(* IEC 61131-3 sources: inproshop/Team-Test5_exported/2.Main, 7 files *)

(* ---- Main.ST ---- *)
(* ==== Generated by PlcOpcUaHmi at 2026-04-27 16:09:01  source=DB80_IO ==== *)
VAR_GLOBAL
	IX8000_0	AT	%IX8000.0:BOOL;
	IX8000_1	AT	%IX8000.1:BOOL;
	IX8000_2	AT	%IX8000.2:BOOL;
	IX8000_3	AT	%IX8000.3:BOOL;
	IX8000_4	AT	%IX8000.4:BOOL;
	IX8000_5	AT	%IX8000.5:BOOL;
	IX8000_6	AT	%IX8000.6:BOOL;
	IX8000_7	AT	%IX8000.7:BOOL;
	IX8001_0_OP08启动按钮HMI1	AT	%IX8001.0:BOOL;
	IX8001_1_OP08停止按钮HMI	AT	%IX8001.1:BOOL;
	IX8001_2_OP08复位按钮HMI	AT	%IX8001.2:BOOL;
	IX8001_3_OP08手自动旋钮HMI	AT	%IX8001.3:BOOL;
	IX8001_4_OP08急停按钮HMI	AT	%IX8001.4:BOOL;
	IX8001_5_OP08启动按钮左	AT	%IX8001.5:BOOL;
	IX8001_6_OP08停止按钮左	AT	%IX8001.6:BOOL;
	IX8001_7_OP08复位按钮左	AT	%IX8001.7:BOOL;
	IX8002_0_OP08手自动旋钮左	AT	%IX8002.0:BOOL;
	IX8002_1_OP08急停按钮左	AT	%IX8002.1:BOOL;
	IX8002_2_OP08启动按钮右	AT	%IX8002.2:BOOL;
	IX8002_3_OP08停止按钮右	AT	%IX8002.3:BOOL;
	IX8002_4_OP08复位按钮右	AT	%IX8002.4:BOOL;
	IX8002_5_OP08手自动旋钮右	AT	%IX8002.5:BOOL;
	IX8002_6_OP08急停按钮右	AT	%IX8002.6:BOOL;
	IX8002_7_OP08安全门1	AT	%IX8002.7:BOOL;
	IX8003_0_OP08安全门2	AT	%IX8003.0:BOOL;
	IX8003_1_OP08安全门3	AT	%IX8003.1:BOOL;
	IX8003_2_OP08安全门4	AT	%IX8003.2:BOOL;
	IX8003_3_OP08安全门5	AT	%IX8003.3:BOOL;
	IX8003_4_OP08安全门6	AT	%IX8003.4:BOOL;
	IX8003_5_OP08安全门7	AT	%IX8003.5:BOOL;
	IX8003_6_OP08安全门8	AT	%IX8003.6:BOOL;
	IX8003_7	AT	%IX8003.7:BOOL;
	IX8004_0	AT	%IX8004.0:BOOL;
	IX8004_1	AT	%IX8004.1:BOOL;
	IX8004_2	AT	%IX8004.2:BOOL;
	IX8004_3	AT	%IX8004.3:BOOL;
	IX8004_4	AT	%IX8004.4:BOOL;
	IX8004_5	AT	%IX8004.5:BOOL;
	IX8004_6	AT	%IX8004.6:BOOL;
	IX8004_7	AT	%IX8004.7:BOOL;
	IX8005_0	AT	%IX8005.0:BOOL;
	IX8005_1	AT	%IX8005.1:BOOL;
	IX8005_2	AT	%IX8005.2:BOOL;
	IX8005_3	AT	%IX8005.3:BOOL;
	IX8005_4	AT	%IX8005.4:BOOL;
	IX8005_5	AT	%IX8005.5:BOOL;
	IX8005_6	AT	%IX8005.6:BOOL;
	IX8005_7	AT	%IX8005.7:BOOL;
	IX8006_0	AT	%IX8006.0:BOOL;
	IX8006_1	AT	%IX8006.1:BOOL;
	IX8006_2	AT	%IX8006.2:BOOL;
	IX8006_3	AT	%IX8006.3:BOOL;
	IX8006_4	AT	%IX8006.4:BOOL;
	IX8006_5	AT	%IX8006.5:BOOL;
	IX8006_6	AT	%IX8006.6:BOOL;
	IX8006_7	AT	%IX8006.7:BOOL;
	IX8007_0	AT	%IX8007.0:BOOL;
	IX8007_1	AT	%IX8007.1:BOOL;
	IX8007_2	AT	%IX8007.2:BOOL;
	IX8007_3	AT	%IX8007.3:BOOL;
	IX8007_4	AT	%IX8007.4:BOOL;
	IX8007_5	AT	%IX8007.5:BOOL;
	IX8007_6	AT	%IX8007.6:BOOL;
	IX8007_7	AT	%IX8007.7:BOOL;
	IX8008_0	AT	%IX8008.0:BOOL;
	IX8008_1	AT	%IX8008.1:BOOL;
	IX8008_2	AT	%IX8008.2:BOOL;
	IX8008_3	AT	%IX8008.3:BOOL;
	IX8008_4	AT	%IX8008.4:BOOL;
	IX8008_5	AT	%IX8008.5:BOOL;
	IX8008_6	AT	%IX8008.6:BOOL;
	IX8008_7	AT	%IX8008.7:BOOL;
	IX8009_0	AT	%IX8009.0:BOOL;
	IX8009_1	AT	%IX8009.1:BOOL;
	IX8009_2	AT	%IX8009.2:BOOL;
	IX8009_3	AT	%IX8009.3:BOOL;
	IX8009_4	AT	%IX8009.4:BOOL;
	IX8009_5	AT	%IX8009.5:BOOL;
	IX8009_6	AT	%IX8009.6:BOOL;
	IX8009_7	AT	%IX8009.7:BOOL;
	IX8100_0_工位1_人工操作按钮	AT	%IX8100.0:BOOL;
	IX8100_1_工位1_物料到位感应Sensor1	AT	%IX8100.1:BOOL;
	IX8100_2_工位1_预留	AT	%IX8100.2:BOOL;
	IX8100_3_工位2_人工操作按钮	AT	%IX8100.3:BOOL;
	IX8100_4_工位2_物料到位感应Sensor2	AT	%IX8100.4:BOOL;
	IX8100_5_工位2_预留	AT	%IX8100.5:BOOL;
	IX8100_6_工位3_人工操作按钮	AT	%IX8100.6:BOOL;
	IX8100_7_工位3_物料到位感应Sensor3	AT	%IX8100.7:BOOL;
	IX8101_0_工位3_预留	AT	%IX8101.0:BOOL;
	IX8101_1_工位4_人工操作按钮	AT	%IX8101.1:BOOL;
	IX8101_2_工位4_物料到位感应Sensor4	AT	%IX8101.2:BOOL;
	IX8101_3_工位4_预留	AT	%IX8101.3:BOOL;
	IX8101_4_工位5_人工操作按钮	AT	%IX8101.4:BOOL;
	IX8101_5_工位5_物料到位感应Sensor5	AT	%IX8101.5:BOOL;
	IX8101_6_工位5_预留	AT	%IX8101.6:BOOL;
	IX8101_7_工位6_人工操作按钮	AT	%IX8101.7:BOOL;
	IX8102_0_工位6_物料到位感应Sensor6	AT	%IX8102.0:BOOL;
	IX8102_1_工位6_预留	AT	%IX8102.1:BOOL;
	IX8102_2_工位7_人工操作按钮	AT	%IX8102.2:BOOL;
	IX8102_3_工位7_物料到位感应Sensor7	AT	%IX8102.3:BOOL;
	IX8102_4_工位7_预留	AT	%IX8102.4:BOOL;
	IX8102_5_工位8_人工操作按钮	AT	%IX8102.5:BOOL;
	IX8102_6_工位8_物料到位感应Sensor8	AT	%IX8102.6:BOOL;
	IX8102_7_工位8_预留	AT	%IX8102.7:BOOL;
	IX8103_0_工位9_人工操作按钮	AT	%IX8103.0:BOOL;
	IX8103_1_工位9_物料到位感应Sensor9	AT	%IX8103.1:BOOL;
	IX8103_2_工位9_预留	AT	%IX8103.2:BOOL;
	IX8103_3_工位10_人工操作按钮	AT	%IX8103.3:BOOL;
	IX8103_4_工位10_物料到位感应Sensor10	AT	%IX8103.4:BOOL;
	IX8103_5_工位10_预留	AT	%IX8103.5:BOOL;
	IX8103_6	AT	%IX8103.6:BOOL;
	IX8103_7	AT	%IX8103.7:BOOL;
	IX8104_0_工位11_人工操作按钮	AT	%IX8104.0:BOOL;
	IX8104_1_工位11_物料到位感应Sensor11	AT	%IX8104.1:BOOL;
	IX8104_2_工位11_预留	AT	%IX8104.2:BOOL;
	IX8104_3_工位12_人工操作按钮	AT	%IX8104.3:BOOL;
	IX8104_4_工位12_物料到位感应Sensor12	AT	%IX8104.4:BOOL;
	IX8104_5_工位12_预留	AT	%IX8104.5:BOOL;
	IX8104_6_工位13_人工操作按钮	AT	%IX8104.6:BOOL;
	IX8104_7_工位13_物料到位感应Sensor13	AT	%IX8104.7:BOOL;
	IX8105_0_工位13_预留	AT	%IX8105.0:BOOL;
	IX8105_1_工位14_人工操作按钮	AT	%IX8105.1:BOOL;
	IX8105_2_工位14_物料到位感应Sensor14	AT	%IX8105.2:BOOL;
	IX8105_3_工位14_预留	AT	%IX8105.3:BOOL;
	IX8105_4_工位15_人工操作按钮	AT	%IX8105.4:BOOL;
	IX8105_5_工位15_物料到位感应Sensor15	AT	%IX8105.5:BOOL;
	IX8105_6_工位15_预留	AT	%IX8105.6:BOOL;
	IX8105_7_工位16_人工操作按钮	AT	%IX8105.7:BOOL;
	IX8106_0_工位16_物料到位感应Sensor16	AT	%IX8106.0:BOOL;
	IX8106_1_工位16_预留	AT	%IX8106.1:BOOL;
	IX8106_2_工位17_人工操作按钮	AT	%IX8106.2:BOOL;
	IX8106_3_工位17_物料到位感应Sensor17	AT	%IX8106.3:BOOL;
	IX8106_4_工位17_预留	AT	%IX8106.4:BOOL;
	IX8106_5_工位18_人工操作按钮	AT	%IX8106.5:BOOL;
	IX8106_6_工位18_物料到位感应Sensor18	AT	%IX8106.6:BOOL;
	IX8106_7_工位18_预留	AT	%IX8106.7:BOOL;
	IX8107_0_工位19_人工操作按钮	AT	%IX8107.0:BOOL;
	IX8107_1_工位19_物料到位感应Sensor19	AT	%IX8107.1:BOOL;
	IX8107_2_工位19_预留	AT	%IX8107.2:BOOL;
	IX8107_3_工位20_人工操作按钮	AT	%IX8107.3:BOOL;
	IX8107_4_工位20_物料到位感应Sensor20	AT	%IX8107.4:BOOL;
	IX8107_5_工位20_预留	AT	%IX8107.5:BOOL;
	IX8107_6	AT	%IX8107.6:BOOL;
	IX8107_7	AT	%IX8107.7:BOOL;
	IX8108_0_工位21_人工操作按钮	AT	%IX8108.0:BOOL;
	IX8108_1_工位21_物料到位感应Sensor21	AT	%IX8108.1:BOOL;
	IX8108_2_工位21_预留	AT	%IX8108.2:BOOL;
	IX8108_3_工位22_人工操作按钮	AT	%IX8108.3:BOOL;
	IX8108_4_工位22_物料到位感应Sensor22	AT	%IX8108.4:BOOL;
	IX8108_5_工位22_预留	AT	%IX8108.5:BOOL;
	IX8108_6_工位23_人工操作按钮	AT	%IX8108.6:BOOL;
	IX8108_7_工位23_物料到位感应Sensor23	AT	%IX8108.7:BOOL;
	IX8109_0_工位23_预留	AT	%IX8109.0:BOOL;
	IX8109_1_工位24_人工操作按钮	AT	%IX8109.1:BOOL;
	IX8109_2_工位24_物料到位感应Sensor24	AT	%IX8109.2:BOOL;
	IX8109_3_工位24_预留	AT	%IX8109.3:BOOL;
	IX8109_4_工位25_人工操作按钮	AT	%IX8109.4:BOOL;
	IX8109_5_工位25_物料到位感应Sensor25	AT	%IX8109.5:BOOL;
	IX8109_6_工位25_预留	AT	%IX8109.6:BOOL;
	IX8109_7_工位26_人工操作按钮	AT	%IX8109.7:BOOL;
	IX8110_0_工位26_物料到位感应Sensor26	AT	%IX8110.0:BOOL;
	IX8110_1_工位26_预留	AT	%IX8110.1:BOOL;
	IX8110_2_工位27_人工操作按钮	AT	%IX8110.2:BOOL;
	IX8110_3_工位27_物料到位感应Sensor27	AT	%IX8110.3:BOOL;
	IX8110_4_工位27_预留	AT	%IX8110.4:BOOL;
	IX8110_5_工位28_人工操作按钮	AT	%IX8110.5:BOOL;
	IX8110_6_工位28_物料到位感应Sensor28	AT	%IX8110.6:BOOL;
	IX8110_7_工位28_预留	AT	%IX8110.7:BOOL;
	IX8111_0_工位29_人工操作按钮	AT	%IX8111.0:BOOL;
	IX8111_1_工位29_物料到位感应Sensor29	AT	%IX8111.1:BOOL;
	IX8111_2_工位29_预留	AT	%IX8111.2:BOOL;
	IX8111_3_工位30_人工操作按钮	AT	%IX8111.3:BOOL;
	IX8111_4_工位30_物料到位感应Sensor30	AT	%IX8111.4:BOOL;
	IX8111_5_工位30_预留1	AT	%IX8111.5:BOOL;
	IX8111_6	AT	%IX8111.6:BOOL;
	IX8111_7	AT	%IX8111.7:BOOL;
	IX8112_0_工位31_人工操作按钮	AT	%IX8112.0:BOOL;
	IX8112_1_工位31_物料到位感应Sensor31	AT	%IX8112.1:BOOL;
	IX8112_2_工位31_预留	AT	%IX8112.2:BOOL;
	IX8112_3_工位32_人工操作按钮	AT	%IX8112.3:BOOL;
	IX8112_4_工位32_物料到位感应Sensor32	AT	%IX8112.4:BOOL;
	IX8112_5_工位32_预留	AT	%IX8112.5:BOOL;
	IX8112_6_工位33_人工操作按钮	AT	%IX8112.6:BOOL;
	IX8112_7_工位33_物料到位感应Sensor33	AT	%IX8112.7:BOOL;
	IX8113_0_工位33_预留	AT	%IX8113.0:BOOL;
	IX8113_1_工位34_人工操作按钮	AT	%IX8113.1:BOOL;
	IX8113_2_工位34_物料到位感应Sensor34	AT	%IX8113.2:BOOL;
	IX8113_3_工位34_预留	AT	%IX8113.3:BOOL;
	IX8113_4_工位35_人工操作按钮	AT	%IX8113.4:BOOL;
	IX8113_5_工位35_物料到位感应Sensor35	AT	%IX8113.5:BOOL;
	IX8113_6_工位35_预留	AT	%IX8113.6:BOOL;
	IX8113_7_工位36_人工操作按钮	AT	%IX8113.7:BOOL;
	IX8114_0_工位36_物料到位感应Sensor36	AT	%IX8114.0:BOOL;
	IX8114_1_工位36_预留	AT	%IX8114.1:BOOL;
	IX8114_2_工位37_人工操作按钮	AT	%IX8114.2:BOOL;
	IX8114_3_工位37_物料到位感应Sensor37	AT	%IX8114.3:BOOL;
	IX8114_4_工位37_预留	AT	%IX8114.4:BOOL;
	IX8114_5_工位38_人工操作按钮	AT	%IX8114.5:BOOL;
	IX8114_6_工位38_物料到位感应Sensor38	AT	%IX8114.6:BOOL;
	IX8114_7_工位38_预留	AT	%IX8114.7:BOOL;
	IX8115_0_工位39_人工操作按钮	AT	%IX8115.0:BOOL;
	IX8115_1_工位39_物料到位感应Sensor39	AT	%IX8115.1:BOOL;
	IX8115_2_工位39_预留	AT	%IX8115.2:BOOL;
	IX8115_3_工位40_人工操作按钮	AT	%IX8115.3:BOOL;
	IX8115_4_工位40_物料到位感应Sensor40	AT	%IX8115.4:BOOL;
	IX8115_5_工位40_预留	AT	%IX8115.5:BOOL;
	IX8115_6	AT	%IX8115.6:BOOL;
	IX8115_7	AT	%IX8115.7:BOOL;
	IX8200_0_工位41_人工操作按钮	AT	%IX8200.0:BOOL;
	IX8200_1_工位41_物料到位感应Sensor41	AT	%IX8200.1:BOOL;
	IX8200_2_工位41_预留	AT	%IX8200.2:BOOL;
	IX8200_3_工位42_人工操作按钮	AT	%IX8200.3:BOOL;
	IX8200_4_工位42_物料到位感应Sensor42	AT	%IX8200.4:BOOL;
	IX8200_5_工位42_预留	AT	%IX8200.5:BOOL;
	IX8200_6_工位43_人工操作按钮	AT	%IX8200.6:BOOL;
	IX8200_7_工位43_物料到位感应Sensor43	AT	%IX8200.7:BOOL;
	IX8201_0_工位43_预留	AT	%IX8201.0:BOOL;
	IX8201_1_工位44_人工操作按钮	AT	%IX8201.1:BOOL;
	IX8201_2_工位44_物料到位感应Sensor44	AT	%IX8201.2:BOOL;
	IX8201_3_工位44_预留	AT	%IX8201.3:BOOL;
	IX8201_4_工位45_人工操作按钮	AT	%IX8201.4:BOOL;
	IX8201_5_工位45_物料到位感应Sensor45	AT	%IX8201.5:BOOL;
	IX8201_6_工位45_预留	AT	%IX8201.6:BOOL;
	IX8201_7_工位46_人工操作按钮	AT	%IX8201.7:BOOL;
	IX8202_0_工位46_物料到位感应Sensor46	AT	%IX8202.0:BOOL;
	IX8202_1_工位46_预留	AT	%IX8202.1:BOOL;
	IX8202_2_工位47_人工操作按钮	AT	%IX8202.2:BOOL;
	IX8202_3_工位47_物料到位感应Sensor47	AT	%IX8202.3:BOOL;
	IX8202_4_工位47_预留	AT	%IX8202.4:BOOL;
	IX8202_5_工位48_人工操作按钮	AT	%IX8202.5:BOOL;
	IX8202_6_工位48_物料到位感应Sensor48	AT	%IX8202.6:BOOL;
	IX8202_7_工位48_预留	AT	%IX8202.7:BOOL;
	IX8203_0_工位49_人工操作按钮	AT	%IX8203.0:BOOL;
	IX8203_1_工位49_物料到位感应Sensor49	AT	%IX8203.1:BOOL;
	IX8203_2_工位49_预留	AT	%IX8203.2:BOOL;
	IX8203_3_工位50_人工操作按钮	AT	%IX8203.3:BOOL;
	IX8203_4_工位50_物料到位感应Sensor50	AT	%IX8203.4:BOOL;
	IX8203_5_工位50_预留	AT	%IX8203.5:BOOL;
	IX8203_6	AT	%IX8203.6:BOOL;
	IX8203_7	AT	%IX8203.7:BOOL;
	IX8204_0_工位51_人工操作按钮	AT	%IX8204.0:BOOL;
	IX8204_1_工位51_物料到位感应Sensor51	AT	%IX8204.1:BOOL;
	IX8204_2_工位51_预留	AT	%IX8204.2:BOOL;
	IX8204_3_工位52_人工操作按钮	AT	%IX8204.3:BOOL;
	IX8204_4_工位52_物料到位感应Sensor52	AT	%IX8204.4:BOOL;
	IX8204_5_工位52_预留	AT	%IX8204.5:BOOL;
	IX8204_6_工位53_人工操作按钮	AT	%IX8204.6:BOOL;
	IX8204_7_工位53_物料到位感应Sensor53	AT	%IX8204.7:BOOL;
	IX8205_0_工位53_预留	AT	%IX8205.0:BOOL;
	IX8205_1_工位54_人工操作按钮	AT	%IX8205.1:BOOL;
	IX8205_2_工位54_物料到位感应Sensor54	AT	%IX8205.2:BOOL;
	IX8205_3_工位54_预留	AT	%IX8205.3:BOOL;
	IX8205_4_工位55_人工操作按钮	AT	%IX8205.4:BOOL;
	IX8205_5_工位55_物料到位感应Sensor55	AT	%IX8205.5:BOOL;
	IX8205_6_工位55_预留	AT	%IX8205.6:BOOL;
	IX8205_7_工位56_人工操作按钮	AT	%IX8205.7:BOOL;
	IX8206_0_工位56_物料到位感应Sensor56	AT	%IX8206.0:BOOL;
	IX8206_1_工位56_预留	AT	%IX8206.1:BOOL;
	IX8206_2_工位57_人工操作按钮	AT	%IX8206.2:BOOL;
	IX8206_3_工位57_物料到位感应Sensor57	AT	%IX8206.3:BOOL;
	IX8206_4_工位57_预留	AT	%IX8206.4:BOOL;
	IX8206_5_工位58_人工操作按钮	AT	%IX8206.5:BOOL;
	IX8206_6_工位58_物料到位感应Sensor58	AT	%IX8206.6:BOOL;
	IX8206_7_工位58_预留	AT	%IX8206.7:BOOL;
	IX8207_0_工位59_人工操作按钮	AT	%IX8207.0:BOOL;
	IX8207_1_工位59_物料到位感应Sensor59	AT	%IX8207.1:BOOL;
	IX8207_2_工位59_预留	AT	%IX8207.2:BOOL;
	IX8207_3_工位60_人工操作按钮	AT	%IX8207.3:BOOL;
	IX8207_4_工位60_物料到位感应Sensor60	AT	%IX8207.4:BOOL;
	IX8207_5_工位60_预留	AT	%IX8207.5:BOOL;
	IX8207_6	AT	%IX8207.6:BOOL;
	IX8207_7	AT	%IX8207.7:BOOL;
	IX8208_0_工位61_人工操作按钮	AT	%IX8208.0:BOOL;
	IX8208_1_工位61_物料到位感应Sensor61	AT	%IX8208.1:BOOL;
	IX8208_2_工位61_预留	AT	%IX8208.2:BOOL;
	IX8208_3_工位62_人工操作按钮	AT	%IX8208.3:BOOL;
	IX8208_4_工位62_物料到位感应Sensor62	AT	%IX8208.4:BOOL;
	IX8208_5_工位62_预留	AT	%IX8208.5:BOOL;
	IX8208_6_工位63_人工操作按钮	AT	%IX8208.6:BOOL;
	IX8208_7_工位63_物料到位感应Sensor63	AT	%IX8208.7:BOOL;
	IX8209_0_工位63_预留	AT	%IX8209.0:BOOL;
	IX8209_1_工位64_人工操作按钮	AT	%IX8209.1:BOOL;
	IX8209_2_工位64_物料到位感应Sensor64	AT	%IX8209.2:BOOL;
	IX8209_3_工位64_预留	AT	%IX8209.3:BOOL;
	IX8209_4_工位65_人工操作按钮	AT	%IX8209.4:BOOL;
	IX8209_5_工位65_物料到位感应Sensor65	AT	%IX8209.5:BOOL;
	IX8209_6_工位65_预留	AT	%IX8209.6:BOOL;
	IX8209_7_工位66_人工操作按钮	AT	%IX8209.7:BOOL;
	IX8210_0_工位66_物料到位感应Sensor66	AT	%IX8210.0:BOOL;
	IX8210_1_工位66_预留	AT	%IX8210.1:BOOL;
	IX8210_2_工位67_人工操作按钮	AT	%IX8210.2:BOOL;
	IX8210_3_工位67_物料到位感应Sensor67	AT	%IX8210.3:BOOL;
	IX8210_4_工位67_预留	AT	%IX8210.4:BOOL;
	IX8210_5_工位68_人工操作按钮	AT	%IX8210.5:BOOL;
	IX8210_6_工位68_物料到位感应Sensor68	AT	%IX8210.6:BOOL;
	IX8210_7_工位68_预留	AT	%IX8210.7:BOOL;
	IX8211_0_工位69_人工操作按钮	AT	%IX8211.0:BOOL;
	IX8211_1_工位69_物料到位感应Sensor69	AT	%IX8211.1:BOOL;
	IX8211_2_工位69_预留	AT	%IX8211.2:BOOL;
	IX8211_3_工位70_人工操作按钮	AT	%IX8211.3:BOOL;
	IX8211_4_工位70_物料到位感应Sensor70	AT	%IX8211.4:BOOL;
	IX8211_5_工位70_预留	AT	%IX8211.5:BOOL;
	IX8211_6	AT	%IX8211.6:BOOL;
	IX8211_7	AT	%IX8211.7:BOOL;
	IX8212_0_工位71_人工操作按钮	AT	%IX8212.0:BOOL;
	IX8212_1_工位71_物料到位感应Sensor71	AT	%IX8212.1:BOOL;
	IX8212_2_工位71_预留	AT	%IX8212.2:BOOL;
	IX8212_3_工位72_人工操作按钮	AT	%IX8212.3:BOOL;
	IX8212_4_工位72_物料到位感应Sensor72	AT	%IX8212.4:BOOL;
	IX8212_5_工位72_预留	AT	%IX8212.5:BOOL;
	IX8212_6_工位73_人工操作按钮	AT	%IX8212.6:BOOL;
	IX8212_7_工位73_物料到位感应Sensor73	AT	%IX8212.7:BOOL;
	IX8213_0_工位73_预留	AT	%IX8213.0:BOOL;
	IX8213_1_工位74_人工操作按钮	AT	%IX8213.1:BOOL;
	IX8213_2_工位74_物料到位感应Sensor74	AT	%IX8213.2:BOOL;
	IX8213_3_工位74_预留	AT	%IX8213.3:BOOL;
	IX8213_4_工位75_人工操作按钮	AT	%IX8213.4:BOOL;
	IX8213_5_工位75_物料到位感应Sensor75	AT	%IX8213.5:BOOL;
	IX8213_6_工位75_预留	AT	%IX8213.6:BOOL;
	IX8213_7_工位76_人工操作按钮	AT	%IX8213.7:BOOL;
	IX8214_0_工位76_物料到位感应Sensor76	AT	%IX8214.0:BOOL;
	IX8214_1_工位76_预留	AT	%IX8214.1:BOOL;
	IX8214_2_工位77_人工操作按钮	AT	%IX8214.2:BOOL;
	IX8214_3_工位77_物料到位感应Sensor77	AT	%IX8214.3:BOOL;
	IX8214_4_工位77_预留	AT	%IX8214.4:BOOL;
	IX8214_5_工位78_人工操作按钮	AT	%IX8214.5:BOOL;
	IX8214_6_工位78_物料到位感应Sensor78	AT	%IX8214.6:BOOL;
	IX8214_7_工位78_预留	AT	%IX8214.7:BOOL;
	IX8215_0_工位79_人工操作按钮	AT	%IX8215.0:BOOL;
	IX8215_1_工位79_物料到位感应Sensor79	AT	%IX8215.1:BOOL;
	IX8215_2_工位79_预留	AT	%IX8215.2:BOOL;
	IX8215_3_工位80_人工操作按钮	AT	%IX8215.3:BOOL;
	IX8215_4_工位80_物料到位感应Sensor80	AT	%IX8215.4:BOOL;
	IX8215_5_工位80_预留	AT	%IX8215.5:BOOL;
	IX8215_6	AT	%IX8215.6:BOOL;
	IX8215_7	AT	%IX8215.7:BOOL;
	IX8300_0_测试1_产品侧边定位气缸CY01_伸出位	AT	%IX8300.0:BOOL;
	IX8300_1_测试1_产品侧边定位气缸CY01_缩回位	AT	%IX8300.1:BOOL;
	IX8300_2_测试1_产品固定气缸CY02_1_锁紧位	AT	%IX8300.2:BOOL;
	IX8300_3_测试1_产品固定气缸CY02_1_松开位	AT	%IX8300.3:BOOL;
	IX8300_4_测试1_产品固定气缸CY02_2_锁紧位	AT	%IX8300.4:BOOL;
	IX8300_5_测试1_产品固定气缸CY02_2_松开位	AT	%IX8300.5:BOOL;
	IX8300_6_测试1_产品封堵A上下气缸CY03_上升位	AT	%IX8300.6:BOOL;
	IX8300_7_测试1_产品封堵A上下气缸CY03_下降位	AT	%IX8300.7:BOOL;
	IX8301_0_测试1_产品封堵A侧推气缸CY04_伸出位	AT	%IX8301.0:BOOL;
	IX8301_1_测试1_产品封堵A侧推气缸CY04_缩回位	AT	%IX8301.1:BOOL;
	IX8301_2_测试1_产品封堵B上下气缸CY05_上升位	AT	%IX8301.2:BOOL;
	IX8301_3_测试1_产品封堵B上下气缸CY05_下降位	AT	%IX8301.3:BOOL;
	IX8301_4_测试1_驱动齿轮气缸CY06_伸出位	AT	%IX8301.4:BOOL;
	IX8301_5_测试1_驱动齿轮气缸CY06_缩回位	AT	%IX8301.5:BOOL;
	IX8301_6_测试1_固定夹爪气缸CY07_夹紧位	AT	%IX8301.6:BOOL;
	IX8301_7_测试1_固定夹爪气缸CY07_缩回位	AT	%IX8301.7:BOOL;
	IX8302_0_测试1_插管测试气缸CY08_上升位	AT	%IX8302.0:BOOL;
	IX8302_1_测试1_插管测试气缸CY08_下降位	AT	%IX8302.1:BOOL;
	IX8302_2_测试1_拔管解扣气缸CY09_上升位	AT	%IX8302.2:BOOL;
	IX8302_3_测试1_拔管解扣气缸CY09_下降位	AT	%IX8302.3:BOOL;
	IX8302_4_缓存NG1_侧边定位气缸CY10_伸出位	AT	%IX8302.4:BOOL;
	IX8302_5_缓存NG1_侧边定位气缸CY10_缩回位	AT	%IX8302.5:BOOL;
	IX8302_6	AT	%IX8302.6:BOOL;
	IX8302_7	AT	%IX8302.7:BOOL;
	IX8303_0_测试1_产品有无检测Sensor101	AT	%IX8303.0:BOOL;
	IX8303_1_测试1_螺杆位置检测Sensor102	AT	%IX8303.1:BOOL;
	IX8303_2_缓存NG1_产品有无检测Sensor103	AT	%IX8303.2:BOOL;
	IX8303_3_测试1_双手启动按钮_左	AT	%IX8303.3:BOOL;
	IX8303_4_测试1_双手启动按钮_右	AT	%IX8303.4:BOOL;
	IX8303_5_测试1_2_急停按钮	AT	%IX8303.5:BOOL;
	IX8303_6_测试1_2_光栅	AT	%IX8303.6:BOOL;
	IX8303_7	AT	%IX8303.7:BOOL;
	IX8304_0_测试2_产品侧边定位气缸CY11_伸出位	AT	%IX8304.0:BOOL;
	IX8304_1_测试2_产品侧边定位气缸CY11_缩回位	AT	%IX8304.1:BOOL;
	IX8304_2_测试2_产品固定气缸CY12_1_锁紧位	AT	%IX8304.2:BOOL;
	IX8304_3_测试2_产品固定气缸CY12_1_松开位	AT	%IX8304.3:BOOL;
	IX8304_4_测试2_产品固定气缸CY12_2_锁紧位	AT	%IX8304.4:BOOL;
	IX8304_5_测试2_产品固定气缸CY12_2_松开位	AT	%IX8304.5:BOOL;
	IX8304_6_测试2_产品封堵A上下气缸CY13_上升位	AT	%IX8304.6:BOOL;
	IX8304_7_测试2_产品封堵A上下气缸CY13_下降位	AT	%IX8304.7:BOOL;
	IX8305_0_测试2_产品封堵A侧推气缸CY14_伸出位	AT	%IX8305.0:BOOL;
	IX8305_1_测试2_产品封堵A侧推气缸CY14_缩回位	AT	%IX8305.1:BOOL;
	IX8305_2_测试2_产品封堵B上下气缸CY15_上升位	AT	%IX8305.2:BOOL;
	IX8305_3_测试2_产品封堵B上下气缸CY15_下降位	AT	%IX8305.3:BOOL;
	IX8305_4_测试2_驱动齿轮气缸CY16_伸出位	AT	%IX8305.4:BOOL;
	IX8305_5_测试2_驱动齿轮气缸CY16_缩回位	AT	%IX8305.5:BOOL;
	IX8305_6_测试2_固定夹爪气缸CY17_夹紧位	AT	%IX8305.6:BOOL;
	IX8305_7_测试2_固定夹爪气缸CY17_缩回位	AT	%IX8305.7:BOOL;
	IX8306_0_测试2_插管测试气缸CY18_上升位	AT	%IX8306.0:BOOL;
	IX8306_1_测试2_插管测试气缸CY18_下降位	AT	%IX8306.1:BOOL;
	IX8306_2_测试2_拔管解扣气缸CY19_上升位	AT	%IX8306.2:BOOL;
	IX8306_3_测试2_拔管解扣气缸CY19_下降位	AT	%IX8306.3:BOOL;
	IX8306_4_缓存NG2_侧边定位气缸CY20_伸出位	AT	%IX8306.4:BOOL;
	IX8306_5_缓存NG2_侧边定位气缸CY20_缩回位	AT	%IX8306.5:BOOL;
	IX8306_6	AT	%IX8306.6:BOOL;
	IX8306_7	AT	%IX8306.7:BOOL;
	IX8307_0_测试2_产品有无检测Sensor111	AT	%IX8307.0:BOOL;
	IX8307_1_测试2_螺杆位置检测Sensor112	AT	%IX8307.1:BOOL;
	IX8307_2_缓存NG2_产品有无检测Sensor113	AT	%IX8307.2:BOOL;
	IX8307_3_测试2_双手启动按钮_左	AT	%IX8307.3:BOOL;
	IX8307_4_测试2_双手启动按钮_右	AT	%IX8307.4:BOOL;
	IX8307_5	AT	%IX8307.5:BOOL;
	IX8307_6	AT	%IX8307.6:BOOL;
	IX8307_7	AT	%IX8307.7:BOOL;
	IX8400_0_测试3_产品侧边定位气缸CY21_伸出位	AT	%IX8400.0:BOOL;
	IX8400_1_测试3_产品侧边定位气缸CY21_缩回位	AT	%IX8400.1:BOOL;
	IX8400_2_测试3_产品固定气缸CY22_1_锁紧位	AT	%IX8400.2:BOOL;
	IX8400_3_测试3_产品固定气缸CY22_1_松开位	AT	%IX8400.3:BOOL;
	IX8400_4_测试3_产品固定气缸CY22_2_锁紧位	AT	%IX8400.4:BOOL;
	IX8400_5_测试3_产品固定气缸CY22_2_松开位	AT	%IX8400.5:BOOL;
	IX8400_6_测试3_产品封堵A上下气缸CY23_上升位	AT	%IX8400.6:BOOL;
	IX8400_7_测试3_产品封堵A上下气缸CY23_下降位	AT	%IX8400.7:BOOL;
	IX8401_0_测试3_产品封堵A侧推气缸CY24_伸出位	AT	%IX8401.0:BOOL;
	IX8401_1_测试3_产品封堵A侧推气缸CY24_缩回位	AT	%IX8401.1:BOOL;
	IX8401_2_测试3_产品封堵B上下气缸CY25_上升位	AT	%IX8401.2:BOOL;
	IX8401_3_测试3_产品封堵B上下气缸CY25_下降位	AT	%IX8401.3:BOOL;
	IX8401_4_测试3_驱动齿轮气缸CY26_伸出位	AT	%IX8401.4:BOOL;
	IX8401_5_测试3_驱动齿轮气缸CY26_缩回位	AT	%IX8401.5:BOOL;
	IX8401_6_测试3_固定夹爪气缸CY27_夹紧位	AT	%IX8401.6:BOOL;
	IX8401_7_测试3_固定夹爪气缸CY27_缩回位	AT	%IX8401.7:BOOL;
	IX8402_0_测试3_插管测试气缸CY28_上升位	AT	%IX8402.0:BOOL;
	IX8402_1_测试3_插管测试气缸CY28_下降位	AT	%IX8402.1:BOOL;
	IX8402_2_测试3_拔管解扣气缸CY29_上升位	AT	%IX8402.2:BOOL;
	IX8402_3_测试3_拔管解扣气缸CY29_下降位	AT	%IX8402.3:BOOL;
	IX8402_4_缓存NG3_侧边定位气缸CY30_伸出位	AT	%IX8402.4:BOOL;
	IX8402_5_缓存NG3_侧边定位气缸CY30_缩回位	AT	%IX8402.5:BOOL;
	IX8402_6	AT	%IX8402.6:BOOL;
	IX8402_7	AT	%IX8402.7:BOOL;
	IX8403_0_测试3_产品有无检测Sensor121	AT	%IX8403.0:BOOL;
	IX8403_1_测试3_螺杆位置检测Sensor122	AT	%IX8403.1:BOOL;
	IX8403_2_缓存NG3_产品有无检测Sensor123	AT	%IX8403.2:BOOL;
	IX8403_3_测试3_双手启动按钮_左	AT	%IX8403.3:BOOL;
	IX8403_4_测试3_双手启动按钮_右	AT	%IX8403.4:BOOL;
	IX8403_5_测试3_4_急停按钮	AT	%IX8403.5:BOOL;
	IX8403_6_测试3_4_光栅	AT	%IX8403.6:BOOL;
	IX8403_7	AT	%IX8403.7:BOOL;
	IX8404_0_测试4_产品侧边定位气缸CY31_伸出位	AT	%IX8404.0:BOOL;
	IX8404_1_测试4_产品侧边定位气缸CY31_缩回位	AT	%IX8404.1:BOOL;
	IX8404_2_测试4_产品固定气缸CY32_1_锁紧位	AT	%IX8404.2:BOOL;
	IX8404_3_测试4_产品固定气缸CY32_1_松开位	AT	%IX8404.3:BOOL;
	IX8404_4_测试4_产品固定气缸CY32_2_锁紧位	AT	%IX8404.4:BOOL;
	IX8404_5_测试4_产品固定气缸CY32_2_松开位	AT	%IX8404.5:BOOL;
	IX8404_6_测试4_产品封堵A上下气缸CY33_上升位	AT	%IX8404.6:BOOL;
	IX8404_7_测试4_产品封堵A上下气缸CY33_下降位	AT	%IX8404.7:BOOL;
	IX8405_0_测试4_产品封堵A侧推气缸CY34_伸出位	AT	%IX8405.0:BOOL;
	IX8405_1_测试4_产品封堵A侧推气缸CY34_缩回位	AT	%IX8405.1:BOOL;
	IX8405_2_测试4_产品封堵B上下气缸CY35_上升位	AT	%IX8405.2:BOOL;
	IX8405_3_测试4_产品封堵B上下气缸CY35_下降位	AT	%IX8405.3:BOOL;
	IX8405_4_测试4_驱动齿轮气缸CY36_伸出位	AT	%IX8405.4:BOOL;
	IX8405_5_测试4_驱动齿轮气缸CY36_缩回位	AT	%IX8405.5:BOOL;
	IX8405_6_测试4_固定夹爪气缸CY37_夹紧位	AT	%IX8405.6:BOOL;
	IX8405_7_测试4_固定夹爪气缸CY37_缩回位	AT	%IX8405.7:BOOL;
	IX8406_0_测试4_插管测试气缸CY38_上升位	AT	%IX8406.0:BOOL;
	IX8406_1_测试4_插管测试气缸CY38_下降位	AT	%IX8406.1:BOOL;
	IX8406_2_测试4_拔管解扣气缸CY39_上升位	AT	%IX8406.2:BOOL;
	IX8406_3_测试4_拔管解扣气缸CY39_下降位	AT	%IX8406.3:BOOL;
	IX8406_4_缓存NG4_侧边定位气缸CY40_伸出位	AT	%IX8406.4:BOOL;
	IX8406_5_缓存NG4_侧边定位气缸CY40_缩回位	AT	%IX8406.5:BOOL;
	IX8406_6	AT	%IX8406.6:BOOL;
	IX8406_7	AT	%IX8406.7:BOOL;
	IX8407_0_测试4_产品有无检测Sensor131	AT	%IX8407.0:BOOL;
	IX8407_1_测试4_螺杆位置检测Sensor132	AT	%IX8407.1:BOOL;
	IX8407_2_缓存NG4_产品有无检测Sensor133	AT	%IX8407.2:BOOL;
	IX8407_3_测试4_双手启动按钮_左	AT	%IX8407.3:BOOL;
	IX8407_4_测试4_双手启动按钮_右	AT	%IX8407.4:BOOL;
	IX8407_5	AT	%IX8407.5:BOOL;
	IX8407_6	AT	%IX8407.6:BOOL;
	IX8407_7	AT	%IX8407.7:BOOL;
	IX8500_0_上料机械手夹爪CY41_夹紧位	AT	%IX8500.0:BOOL;
	IX8500_1_上料机械手夹爪CY41_打开位	AT	%IX8500.1:BOOL;
	IX8500_2_上料机械手夹爪物料有无检测Sensor141	AT	%IX8500.2:BOOL;
	IX8500_3	AT	%IX8500.3:BOOL;
	IX8500_4	AT	%IX8500.4:BOOL;
	IX8500_5	AT	%IX8500.5:BOOL;
	IX8500_6	AT	%IX8500.6:BOOL;
	IX8500_7	AT	%IX8500.7:BOOL;
	IX8501_0	AT	%IX8501.0:BOOL;
	IX8501_1	AT	%IX8501.1:BOOL;
	IX8501_2	AT	%IX8501.2:BOOL;
	IX8501_3	AT	%IX8501.3:BOOL;
	IX8501_4	AT	%IX8501.4:BOOL;
	IX8501_5	AT	%IX8501.5:BOOL;
	IX8501_6	AT	%IX8501.6:BOOL;
	IX8501_7	AT	%IX8501.7:BOOL;
	IX8600_0_码垛机械手夹爪CY45_夹紧位	AT	%IX8600.0:BOOL;
	IX8600_1_码垛机械手夹爪CY45_打开位	AT	%IX8600.1:BOOL;
	IX8600_2_码垛机械手隔板真空吸Vac01_真空表头	AT	%IX8600.2:BOOL;
	IX8600_3	AT	%IX8600.3:BOOL;
	IX8600_4	AT	%IX8600.4:BOOL;
	IX8600_5	AT	%IX8600.5:BOOL;
	IX8600_6	AT	%IX8600.6:BOOL;
	IX8600_7	AT	%IX8600.7:BOOL;
	IX8601_0_码垛机械手夹爪物料有无检测Sensor145	AT	%IX8601.0:BOOL;
	IX8601_1_码垛机械手夹爪隔板取料检测Sensor146	AT	%IX8601.1:BOOL;
	IX8601_2_码垛机械手夹爪隔板取料检测Sensor147	AT	%IX8601.2:BOOL;
	IX8601_3	AT	%IX8601.3:BOOL;
	IX8601_4	AT	%IX8601.4:BOOL;
	IX8601_5	AT	%IX8601.5:BOOL;
	IX8601_6	AT	%IX8601.6:BOOL;
	IX8601_7	AT	%IX8601.7:BOOL;
	IX8700_0_NG流线放料位有无检测Sensor151	AT	%IX8700.0:BOOL;
	IX8700_1_NG流线位移到位检测Sensor152	AT	%IX8700.1:BOOL;
	IX8700_2_NG流线满料检测Sensor153	AT	%IX8700.2:BOOL;
	IX8700_3_码垛区域1托盘到位检测	AT	%IX8700.3:BOOL;
	IX8700_4_码垛区域1安全光栅	AT	%IX8700.4:BOOL;
	IX8700_5_码垛区域1上托盘请求	AT	%IX8700.5:BOOL;
	IX8700_6_码垛区域1下托盘请求	AT	%IX8700.6:BOOL;
	IX8700_7_码垛区域2托盘到位检测	AT	%IX8700.7:BOOL;
	IX8701_0_码垛区域2安全光栅	AT	%IX8701.0:BOOL;
	IX8701_1_码垛区域2上托盘请求	AT	%IX8701.1:BOOL;
	IX8701_2_码垛区域2下托盘请求	AT	%IX8701.2:BOOL;
	IX8701_3_码垛区域3托盘到位检测	AT	%IX8701.3:BOOL;
	IX8701_4_码垛区域3安全光栅	AT	%IX8701.4:BOOL;
	IX8701_5_码垛区域3上托盘请求	AT	%IX8701.5:BOOL;
	IX8701_6_码垛区域3下托盘请求	AT	%IX8701.6:BOOL;
	IX8701_7	AT	%IX8701.7:BOOL;
	QX8000_0	AT	%QX8000.0:BOOL;
	QX8000_1	AT	%QX8000.1:BOOL;
	QX8000_2	AT	%QX8000.2:BOOL;
	QX8000_3	AT	%QX8000.3:BOOL;
	QX8000_4	AT	%QX8000.4:BOOL;
	QX8000_5	AT	%QX8000.5:BOOL;
	QX8000_6	AT	%QX8000.6:BOOL;
	QX8000_7	AT	%QX8000.7:BOOL;
	QX8001_0_OP08启动按钮指示灯HMI	AT	%QX8001.0:BOOL;
	QX8001_1_OP08停止按钮指示灯HMI	AT	%QX8001.1:BOOL;
	QX8001_2_OP08复位按钮指示灯HMI	AT	%QX8001.2:BOOL;
	QX8001_3_OP08启动按钮指示灯左	AT	%QX8001.3:BOOL;
	QX8001_4_OP08停止按钮指示灯左	AT	%QX8001.4:BOOL;
	QX8001_5_OP08复位按钮指示灯左	AT	%QX8001.5:BOOL;
	QX8001_6_OP08启动按钮指示灯右	AT	%QX8001.6:BOOL;
	QX8001_7_OP08停止按钮指示灯右	AT	%QX8001.7:BOOL;
	QX8002_0_OP08复位按钮指示灯右	AT	%QX8002.0:BOOL;
	QX8002_1_OP08三色灯红	AT	%QX8002.1:BOOL;
	QX8002_2_OP08三色灯黄	AT	%QX8002.2:BOOL;
	QX8002_3_OP08三色灯绿	AT	%QX8002.3:BOOL;
	QX8002_4_OP08蜂鸣器	AT	%QX8002.4:BOOL;
	QX8002_5_OP08照明灯	AT	%QX8002.5:BOOL;
	QX8002_6_机械手急停控制继电器	AT	%QX8002.6:BOOL;
	QX8002_7_机械手安全门控制继电器	AT	%QX8002.7:BOOL;
	QX8003_0	AT	%QX8003.0:BOOL;
	QX8003_1	AT	%QX8003.1:BOOL;
	QX8003_2	AT	%QX8003.2:BOOL;
	QX8003_3	AT	%QX8003.3:BOOL;
	QX8003_4	AT	%QX8003.4:BOOL;
	QX8003_5	AT	%QX8003.5:BOOL;
	QX8003_6	AT	%QX8003.6:BOOL;
	QX8003_7	AT	%QX8003.7:BOOL;
	QX8004_0	AT	%QX8004.0:BOOL;
	QX8004_1	AT	%QX8004.1:BOOL;
	QX8004_2	AT	%QX8004.2:BOOL;
	QX8004_3	AT	%QX8004.3:BOOL;
	QX8004_4	AT	%QX8004.4:BOOL;
	QX8004_5	AT	%QX8004.5:BOOL;
	QX8004_6	AT	%QX8004.6:BOOL;
	QX8004_7	AT	%QX8004.7:BOOL;
	QX8005_0	AT	%QX8005.0:BOOL;
	QX8005_1	AT	%QX8005.1:BOOL;
	QX8005_2	AT	%QX8005.2:BOOL;
	QX8005_3	AT	%QX8005.3:BOOL;
	QX8005_4	AT	%QX8005.4:BOOL;
	QX8005_5	AT	%QX8005.5:BOOL;
	QX8005_6	AT	%QX8005.6:BOOL;
	QX8005_7	AT	%QX8005.7:BOOL;
	QX8006_0	AT	%QX8006.0:BOOL;
	QX8006_1	AT	%QX8006.1:BOOL;
	QX8006_2	AT	%QX8006.2:BOOL;
	QX8006_3	AT	%QX8006.3:BOOL;
	QX8006_4	AT	%QX8006.4:BOOL;
	QX8006_5	AT	%QX8006.5:BOOL;
	QX8006_6	AT	%QX8006.6:BOOL;
	QX8006_7	AT	%QX8006.7:BOOL;
	QX8007_0	AT	%QX8007.0:BOOL;
	QX8007_1	AT	%QX8007.1:BOOL;
	QX8007_2	AT	%QX8007.2:BOOL;
	QX8007_3	AT	%QX8007.3:BOOL;
	QX8007_4	AT	%QX8007.4:BOOL;
	QX8007_5	AT	%QX8007.5:BOOL;
	QX8007_6	AT	%QX8007.6:BOOL;
	QX8007_7	AT	%QX8007.7:BOOL;
	QX8008_0	AT	%QX8008.0:BOOL;
	QX8008_1	AT	%QX8008.1:BOOL;
	QX8008_2	AT	%QX8008.2:BOOL;
	QX8008_3	AT	%QX8008.3:BOOL;
	QX8008_4	AT	%QX8008.4:BOOL;
	QX8008_5	AT	%QX8008.5:BOOL;
	QX8008_6	AT	%QX8008.6:BOOL;
	QX8008_7	AT	%QX8008.7:BOOL;
	QX8009_0	AT	%QX8009.0:BOOL;
	QX8009_1	AT	%QX8009.1:BOOL;
	QX8009_2	AT	%QX8009.2:BOOL;
	QX8009_3	AT	%QX8009.3:BOOL;
	QX8009_4	AT	%QX8009.4:BOOL;
	QX8009_5	AT	%QX8009.5:BOOL;
	QX8009_6	AT	%QX8009.6:BOOL;
	QX8009_7	AT	%QX8009.7:BOOL;
	QX8100_0_工位1_指示灯_红	AT	%QX8100.0:BOOL;
	QX8100_1_工位1_指示灯_黄	AT	%QX8100.1:BOOL;
	QX8100_2_工位1_指示灯_绿	AT	%QX8100.2:BOOL;
	QX8100_3_工位1_上电机正转	AT	%QX8100.3:BOOL;
	QX8100_4_工位1_上电机反转	AT	%QX8100.4:BOOL;
	QX8100_5_工位1_下电机正转	AT	%QX8100.5:BOOL;
	QX8100_6_工位1_下电机反转	AT	%QX8100.6:BOOL;
	QX8100_7_工位1_5开关电源控制	AT	%QX8100.7:BOOL;
	QX8101_0_工位2_指示灯_红	AT	%QX8101.0:BOOL;
	QX8101_1_工位2_指示灯_黄	AT	%QX8101.1:BOOL;
	QX8101_2_工位2_指示灯_绿	AT	%QX8101.2:BOOL;
	QX8101_3_工位2_上电机正转	AT	%QX8101.3:BOOL;
	QX8101_4_工位2_上电机反转	AT	%QX8101.4:BOOL;
	QX8101_5_工位2_下电机正转	AT	%QX8101.5:BOOL;
	QX8101_6_工位2_下电机反转	AT	%QX8101.6:BOOL;
	QX8101_7_工位2_预留	AT	%QX8101.7:BOOL;
	QX8102_0_工位3_指示灯_红	AT	%QX8102.0:BOOL;
	QX8102_1_工位3_指示灯_黄	AT	%QX8102.1:BOOL;
	QX8102_2_工位3_指示灯_绿	AT	%QX8102.2:BOOL;
	QX8102_3_工位3_上电机正转	AT	%QX8102.3:BOOL;
	QX8102_4_工位3_上电机反转	AT	%QX8102.4:BOOL;
	QX8102_5_工位3_下电机正转	AT	%QX8102.5:BOOL;
	QX8102_6_工位3_下电机反转	AT	%QX8102.6:BOOL;
	QX8102_7_工位3_预留	AT	%QX8102.7:BOOL;
	QX8103_0_工位4_指示灯_红	AT	%QX8103.0:BOOL;
	QX8103_1_工位4_指示灯_黄	AT	%QX8103.1:BOOL;
	QX8103_2_工位4_指示灯_绿	AT	%QX8103.2:BOOL;
	QX8103_3_工位4_上电机正转	AT	%QX8103.3:BOOL;
	QX8103_4_工位4_上电机反转	AT	%QX8103.4:BOOL;
	QX8103_5_工位4_下电机正转	AT	%QX8103.5:BOOL;
	QX8103_6_工位4_下电机反转	AT	%QX8103.6:BOOL;
	QX8103_7_工位4_预留	AT	%QX8103.7:BOOL;
	QX8104_0_工位5_指示灯_红	AT	%QX8104.0:BOOL;
	QX8104_1_工位5_指示灯_黄	AT	%QX8104.1:BOOL;
	QX8104_2_工位5_指示灯_绿	AT	%QX8104.2:BOOL;
	QX8104_3_工位5_上电机正转	AT	%QX8104.3:BOOL;
	QX8104_4_工位5_上电机反转	AT	%QX8104.4:BOOL;
	QX8104_5_工位5_下电机正转	AT	%QX8104.5:BOOL;
	QX8104_6_工位5_下电机反转	AT	%QX8104.6:BOOL;
	QX8104_7_工位5_预留	AT	%QX8104.7:BOOL;
	QX8105_0_工位6_指示灯_红	AT	%QX8105.0:BOOL;
	QX8105_1_工位6_指示灯_黄	AT	%QX8105.1:BOOL;
	QX8105_2_工位6_指示灯_绿	AT	%QX8105.2:BOOL;
	QX8105_3_工位6_上电机正转	AT	%QX8105.3:BOOL;
	QX8105_4_工位6_上电机反转	AT	%QX8105.4:BOOL;
	QX8105_5_工位6_下电机正转	AT	%QX8105.5:BOOL;
	QX8105_6_工位6_下电机反转	AT	%QX8105.6:BOOL;
	QX8105_7_工位6_10开关电源控制	AT	%QX8105.7:BOOL;
	QX8106_0_工位7_指示灯_红	AT	%QX8106.0:BOOL;
	QX8106_1_工位7_指示灯_黄	AT	%QX8106.1:BOOL;
	QX8106_2_工位7_指示灯_绿	AT	%QX8106.2:BOOL;
	QX8106_3_工位7_上电机正转	AT	%QX8106.3:BOOL;
	QX8106_4_工位7_上电机反转	AT	%QX8106.4:BOOL;
	QX8106_5_工位7_下电机正转	AT	%QX8106.5:BOOL;
	QX8106_6_工位7_下电机反转	AT	%QX8106.6:BOOL;
	QX8106_7_工位7_预留	AT	%QX8106.7:BOOL;
	QX8107_0_工位8_指示灯_红	AT	%QX8107.0:BOOL;
	QX8107_1_工位8_指示灯_黄	AT	%QX8107.1:BOOL;
	QX8107_2_工位8_指示灯_绿	AT	%QX8107.2:BOOL;
	QX8107_3_工位8_上电机正转	AT	%QX8107.3:BOOL;
	QX8107_4_工位8_上电机反转	AT	%QX8107.4:BOOL;
	QX8107_5_工位8_下电机正转	AT	%QX8107.5:BOOL;
	QX8107_6_工位8_下电机反转	AT	%QX8107.6:BOOL;
	QX8107_7_工位8_预留	AT	%QX8107.7:BOOL;
	QX8108_0_工位9_指示灯_红	AT	%QX8108.0:BOOL;
	QX8108_1_工位9_指示灯_黄	AT	%QX8108.1:BOOL;
	QX8108_2_工位9_指示灯_绿	AT	%QX8108.2:BOOL;
	QX8108_3_工位9_上电机正转	AT	%QX8108.3:BOOL;
	QX8108_4_工位9_上电机反转	AT	%QX8108.4:BOOL;
	QX8108_5_工位9_下电机正转	AT	%QX8108.5:BOOL;
	QX8108_6_工位9_下电机反转	AT	%QX8108.6:BOOL;
	QX8108_7_工位9_预留	AT	%QX8108.7:BOOL;
	QX8109_0_工位10_指示灯_红	AT	%QX8109.0:BOOL;
	QX8109_1_工位10_指示灯_黄	AT	%QX8109.1:BOOL;
	QX8109_2_工位10_指示灯_绿	AT	%QX8109.2:BOOL;
	QX8109_3_工位10_上电机正转	AT	%QX8109.3:BOOL;
	QX8109_4_工位10_上电机反转	AT	%QX8109.4:BOOL;
	QX8109_5_工位10_下电机正转	AT	%QX8109.5:BOOL;
	QX8109_6_工位10_下电机反转	AT	%QX8109.6:BOOL;
	QX8109_7_工位10_预留	AT	%QX8109.7:BOOL;
	QX8110_0_工位11_指示灯_红	AT	%QX8110.0:BOOL;
	QX8110_1_工位11_指示灯_黄	AT	%QX8110.1:BOOL;
	QX8110_2_工位11_指示灯_绿	AT	%QX8110.2:BOOL;
	QX8110_3_工位11_上电机正转	AT	%QX8110.3:BOOL;
	QX8110_4_工位11_上电机反转	AT	%QX8110.4:BOOL;
	QX8110_5_工位11_下电机正转	AT	%QX8110.5:BOOL;
	QX8110_6_工位11_下电机反转	AT	%QX8110.6:BOOL;
	QX8110_7_工位11_15开关电源控制	AT	%QX8110.7:BOOL;
	QX8111_0_工位12_指示灯_红	AT	%QX8111.0:BOOL;
	QX8111_1_工位12_指示灯_黄	AT	%QX8111.1:BOOL;
	QX8111_2_工位12_指示灯_绿	AT	%QX8111.2:BOOL;
	QX8111_3_工位12_上电机正转	AT	%QX8111.3:BOOL;
	QX8111_4_工位12_上电机反转	AT	%QX8111.4:BOOL;
	QX8111_5_工位12_下电机正转	AT	%QX8111.5:BOOL;
	QX8111_6_工位12_下电机反转	AT	%QX8111.6:BOOL;
	QX8111_7_工位12_预留	AT	%QX8111.7:BOOL;
	QX8112_0_工位13_指示灯_红	AT	%QX8112.0:BOOL;
	QX8112_1_工位13_指示灯_黄	AT	%QX8112.1:BOOL;
	QX8112_2_工位13_指示灯_绿	AT	%QX8112.2:BOOL;
	QX8112_3_工位13_上电机正转	AT	%QX8112.3:BOOL;
	QX8112_4_工位13_上电机反转	AT	%QX8112.4:BOOL;
	QX8112_5_工位13_下电机正转	AT	%QX8112.5:BOOL;
	QX8112_6_工位13_下电机反转	AT	%QX8112.6:BOOL;
	QX8112_7_工位13_预留	AT	%QX8112.7:BOOL;
	QX8113_0_工位14_指示灯_红	AT	%QX8113.0:BOOL;
	QX8113_1_工位14_指示灯_黄	AT	%QX8113.1:BOOL;
	QX8113_2_工位14_指示灯_绿	AT	%QX8113.2:BOOL;
	QX8113_3_工位14_上电机正转	AT	%QX8113.3:BOOL;
	QX8113_4_工位14_上电机反转	AT	%QX8113.4:BOOL;
	QX8113_5_工位14_下电机正转	AT	%QX8113.5:BOOL;
	QX8113_6_工位14_下电机反转	AT	%QX8113.6:BOOL;
	QX8113_7_工位14_预留	AT	%QX8113.7:BOOL;
	QX8114_0_工位15_指示灯_红	AT	%QX8114.0:BOOL;
	QX8114_1_工位15_指示灯_黄	AT	%QX8114.1:BOOL;
	QX8114_2_工位15_指示灯_绿	AT	%QX8114.2:BOOL;
	QX8114_3_工位15_上电机正转	AT	%QX8114.3:BOOL;
	QX8114_4_工位15_上电机反转	AT	%QX8114.4:BOOL;
	QX8114_5_工位15_下电机正转	AT	%QX8114.5:BOOL;
	QX8114_6_工位15_下电机反转	AT	%QX8114.6:BOOL;
	QX8114_7_工位15_预留	AT	%QX8114.7:BOOL;
	QX8115_0_工位16_指示灯_红	AT	%QX8115.0:BOOL;
	QX8115_1_工位16_指示灯_黄	AT	%QX8115.1:BOOL;
	QX8115_2_工位16_指示灯_绿	AT	%QX8115.2:BOOL;
	QX8115_3_工位16_上电机正转	AT	%QX8115.3:BOOL;
	QX8115_4_工位16_上电机反转	AT	%QX8115.4:BOOL;
	QX8115_5_工位16_下电机正转	AT	%QX8115.5:BOOL;
	QX8115_6_工位16_下电机反转	AT	%QX8115.6:BOOL;
	QX8115_7_工位16_20开关电源控制	AT	%QX8115.7:BOOL;
	QX8116_0_工位17_指示灯_红	AT	%QX8116.0:BOOL;
	QX8116_1_工位17_指示灯_黄	AT	%QX8116.1:BOOL;
	QX8116_2_工位17_指示灯_绿	AT	%QX8116.2:BOOL;
	QX8116_3_工位17_上电机正转	AT	%QX8116.3:BOOL;
	QX8116_4_工位17_上电机反转	AT	%QX8116.4:BOOL;
	QX8116_5_工位17_下电机正转	AT	%QX8116.5:BOOL;
	QX8116_6_工位17_下电机反转	AT	%QX8116.6:BOOL;
	QX8116_7_工位17_预留	AT	%QX8116.7:BOOL;
	QX8117_0_工位18_指示灯_红	AT	%QX8117.0:BOOL;
	QX8117_1_工位18_指示灯_黄	AT	%QX8117.1:BOOL;
	QX8117_2_工位18_指示灯_绿	AT	%QX8117.2:BOOL;
	QX8117_3_工位18_上电机正转	AT	%QX8117.3:BOOL;
	QX8117_4_工位18_上电机反转	AT	%QX8117.4:BOOL;
	QX8117_5_工位18_下电机正转	AT	%QX8117.5:BOOL;
	QX8117_6_工位18_下电机反转	AT	%QX8117.6:BOOL;
	QX8117_7_工位18_预留	AT	%QX8117.7:BOOL;
	QX8118_0_工位19_指示灯_红	AT	%QX8118.0:BOOL;
	QX8118_1_工位19_指示灯_黄	AT	%QX8118.1:BOOL;
	QX8118_2_工位19_指示灯_绿	AT	%QX8118.2:BOOL;
	QX8118_3_工位19_上电机正转	AT	%QX8118.3:BOOL;
	QX8118_4_工位19_上电机反转	AT	%QX8118.4:BOOL;
	QX8118_5_工位19_下电机正转	AT	%QX8118.5:BOOL;
	QX8118_6_工位19_下电机反转	AT	%QX8118.6:BOOL;
	QX8118_7_工位19_预留	AT	%QX8118.7:BOOL;
	QX8119_0_工位20_指示灯_红	AT	%QX8119.0:BOOL;
	QX8119_1_工位20_指示灯_黄	AT	%QX8119.1:BOOL;
	QX8119_2_工位20_指示灯_绿	AT	%QX8119.2:BOOL;
	QX8119_3_工位20_上电机正转	AT	%QX8119.3:BOOL;
	QX8119_4_工位20_上电机反转	AT	%QX8119.4:BOOL;
	QX8119_5_工位20_下电机正转	AT	%QX8119.5:BOOL;
	QX8119_6_工位20_下电机反转	AT	%QX8119.6:BOOL;
	QX8119_7_工位20_预留	AT	%QX8119.7:BOOL;
	QX8120_0_工位21_指示灯_红	AT	%QX8120.0:BOOL;
	QX8120_1_工位21_指示灯_黄	AT	%QX8120.1:BOOL;
	QX8120_2_工位21_指示灯_绿	AT	%QX8120.2:BOOL;
	QX8120_3_工位21_上电机正转	AT	%QX8120.3:BOOL;
	QX8120_4_工位21_上电机反转	AT	%QX8120.4:BOOL;
	QX8120_5_工位21_下电机正转	AT	%QX8120.5:BOOL;
	QX8120_6_工位21_下电机反转	AT	%QX8120.6:BOOL;
	QX8120_7_工位21_25开关电源控制	AT	%QX8120.7:BOOL;
	QX8121_0_工位22_指示灯_红	AT	%QX8121.0:BOOL;
	QX8121_1_工位22_指示灯_黄	AT	%QX8121.1:BOOL;
	QX8121_2_工位22_指示灯_绿	AT	%QX8121.2:BOOL;
	QX8121_3_工位22_上电机正转	AT	%QX8121.3:BOOL;
	QX8121_4_工位22_上电机反转	AT	%QX8121.4:BOOL;
	QX8121_5_工位22_下电机正转	AT	%QX8121.5:BOOL;
	QX8121_6_工位22_下电机反转	AT	%QX8121.6:BOOL;
	QX8121_7_工位22_预留	AT	%QX8121.7:BOOL;
	QX8122_0_工位23_指示灯_红	AT	%QX8122.0:BOOL;
	QX8122_1_工位23_指示灯_黄	AT	%QX8122.1:BOOL;
	QX8122_2_工位23_指示灯_绿	AT	%QX8122.2:BOOL;
	QX8122_3_工位23_上电机正转	AT	%QX8122.3:BOOL;
	QX8122_4_工位23_上电机反转	AT	%QX8122.4:BOOL;
	QX8122_5_工位23_下电机正转	AT	%QX8122.5:BOOL;
	QX8122_6_工位23_下电机反转	AT	%QX8122.6:BOOL;
	QX8122_7_工位23_预留	AT	%QX8122.7:BOOL;
	QX8123_0_工位24_指示灯_红	AT	%QX8123.0:BOOL;
	QX8123_1_工位24_指示灯_黄	AT	%QX8123.1:BOOL;
	QX8123_2_工位24_指示灯_绿	AT	%QX8123.2:BOOL;
	QX8123_3_工位24_上电机正转	AT	%QX8123.3:BOOL;
	QX8123_4_工位24_上电机反转	AT	%QX8123.4:BOOL;
	QX8123_5_工位24_下电机正转	AT	%QX8123.5:BOOL;
	QX8123_6_工位24_下电机反转	AT	%QX8123.6:BOOL;
	QX8123_7_工位24_预留	AT	%QX8123.7:BOOL;
	QX8124_0_工位25_指示灯_红	AT	%QX8124.0:BOOL;
	QX8124_1_工位25_指示灯_黄	AT	%QX8124.1:BOOL;
	QX8124_2_工位25_指示灯_绿	AT	%QX8124.2:BOOL;
	QX8124_3_工位25_上电机正转	AT	%QX8124.3:BOOL;
	QX8124_4_工位25_上电机反转	AT	%QX8124.4:BOOL;
	QX8124_5_工位25_下电机正转	AT	%QX8124.5:BOOL;
	QX8124_6_工位25_下电机反转	AT	%QX8124.6:BOOL;
	QX8124_7_工位25_预留	AT	%QX8124.7:BOOL;
	QX8125_0_工位26_指示灯_红	AT	%QX8125.0:BOOL;
	QX8125_1_工位26_指示灯_黄	AT	%QX8125.1:BOOL;
	QX8125_2_工位26_指示灯_绿	AT	%QX8125.2:BOOL;
	QX8125_3_工位26_上电机正转	AT	%QX8125.3:BOOL;
	QX8125_4_工位26_上电机反转	AT	%QX8125.4:BOOL;
	QX8125_5_工位26_下电机正转	AT	%QX8125.5:BOOL;
	QX8125_6_工位26_下电机反转	AT	%QX8125.6:BOOL;
	QX8125_7_工位26_30开关电源控制	AT	%QX8125.7:BOOL;
	QX8126_0_工位27_指示灯_红	AT	%QX8126.0:BOOL;
	QX8126_1_工位27_指示灯_黄	AT	%QX8126.1:BOOL;
	QX8126_2_工位27_指示灯_绿	AT	%QX8126.2:BOOL;
	QX8126_3_工位27_上电机正转	AT	%QX8126.3:BOOL;
	QX8126_4_工位27_上电机反转	AT	%QX8126.4:BOOL;
	QX8126_5_工位27_下电机正转	AT	%QX8126.5:BOOL;
	QX8126_6_工位27_下电机反转	AT	%QX8126.6:BOOL;
	QX8126_7_工位27_预留	AT	%QX8126.7:BOOL;
	QX8127_0_工位28_指示灯_红	AT	%QX8127.0:BOOL;
	QX8127_1_工位28_指示灯_黄	AT	%QX8127.1:BOOL;
	QX8127_2_工位28_指示灯_绿	AT	%QX8127.2:BOOL;
	QX8127_3_工位28_上电机正转	AT	%QX8127.3:BOOL;
	QX8127_4_工位28_上电机反转	AT	%QX8127.4:BOOL;
	QX8127_5_工位28_下电机正转	AT	%QX8127.5:BOOL;
	QX8127_6_工位28_下电机反转	AT	%QX8127.6:BOOL;
	QX8127_7_工位28_预留	AT	%QX8127.7:BOOL;
	QX8128_0_工位29_指示灯_红	AT	%QX8128.0:BOOL;
	QX8128_1_工位29_指示灯_黄	AT	%QX8128.1:BOOL;
	QX8128_2_工位29_指示灯_绿	AT	%QX8128.2:BOOL;
	QX8128_3_工位29_上电机正转	AT	%QX8128.3:BOOL;
	QX8128_4_工位29_上电机反转	AT	%QX8128.4:BOOL;
	QX8128_5_工位29_下电机正转	AT	%QX8128.5:BOOL;
	QX8128_6_工位29_下电机反转	AT	%QX8128.6:BOOL;
	QX8128_7_工位29_预留	AT	%QX8128.7:BOOL;
	QX8129_0_工位30_指示灯_红	AT	%QX8129.0:BOOL;
	QX8129_1_工位30_指示灯_黄	AT	%QX8129.1:BOOL;
	QX8129_2_工位30_指示灯_绿	AT	%QX8129.2:BOOL;
	QX8129_3_工位30_上电机正转	AT	%QX8129.3:BOOL;
	QX8129_4_工位30_上电机反转	AT	%QX8129.4:BOOL;
	QX8129_5_工位30_下电机正转	AT	%QX8129.5:BOOL;
	QX8129_6_工位30_下电机反转	AT	%QX8129.6:BOOL;
	QX8129_7_工位30_预留	AT	%QX8129.7:BOOL;
	QX8130_0_工位31_指示灯_红	AT	%QX8130.0:BOOL;
	QX8130_1_工位31_指示灯_黄	AT	%QX8130.1:BOOL;
	QX8130_2_工位31_指示灯_绿	AT	%QX8130.2:BOOL;
	QX8130_3_工位31_上电机正转	AT	%QX8130.3:BOOL;
	QX8130_4_工位31_上电机反转	AT	%QX8130.4:BOOL;
	QX8130_5_工位31_下电机正转	AT	%QX8130.5:BOOL;
	QX8130_6_工位31_下电机反转	AT	%QX8130.6:BOOL;
	QX8130_7_工位31_35开关电源控制	AT	%QX8130.7:BOOL;
	QX8131_0_工位32_指示灯_红	AT	%QX8131.0:BOOL;
	QX8131_1_工位32_指示灯_黄	AT	%QX8131.1:BOOL;
	QX8131_2_工位32_指示灯_绿	AT	%QX8131.2:BOOL;
	QX8131_3_工位32_上电机正转	AT	%QX8131.3:BOOL;
	QX8131_4_工位32_上电机反转	AT	%QX8131.4:BOOL;
	QX8131_5_工位32_下电机正转	AT	%QX8131.5:BOOL;
	QX8131_6_工位32_下电机反转	AT	%QX8131.6:BOOL;
	QX8131_7_工位32_预留	AT	%QX8131.7:BOOL;
	QX8132_0_工位33_指示灯_红	AT	%QX8132.0:BOOL;
	QX8132_1_工位33_指示灯_黄	AT	%QX8132.1:BOOL;
	QX8132_2_工位33_指示灯_绿	AT	%QX8132.2:BOOL;
	QX8132_3_工位33_上电机正转	AT	%QX8132.3:BOOL;
	QX8132_4_工位33_上电机反转	AT	%QX8132.4:BOOL;
	QX8132_5_工位33_下电机正转	AT	%QX8132.5:BOOL;
	QX8132_6_工位33_下电机反转	AT	%QX8132.6:BOOL;
	QX8132_7_工位33_预留	AT	%QX8132.7:BOOL;
	QX8133_0_工位34_指示灯_红	AT	%QX8133.0:BOOL;
	QX8133_1_工位34_指示灯_黄	AT	%QX8133.1:BOOL;
	QX8133_2_工位34_指示灯_绿	AT	%QX8133.2:BOOL;
	QX8133_3_工位34_上电机正转	AT	%QX8133.3:BOOL;
	QX8133_4_工位34_上电机反转	AT	%QX8133.4:BOOL;
	QX8133_5_工位34_下电机正转	AT	%QX8133.5:BOOL;
	QX8133_6_工位34_下电机反转	AT	%QX8133.6:BOOL;
	QX8133_7_工位34_预留	AT	%QX8133.7:BOOL;
	QX8134_0_工位35_指示灯_红	AT	%QX8134.0:BOOL;
	QX8134_1_工位35_指示灯_黄	AT	%QX8134.1:BOOL;
	QX8134_2_工位35_指示灯_绿	AT	%QX8134.2:BOOL;
	QX8134_3_工位35_上电机正转	AT	%QX8134.3:BOOL;
	QX8134_4_工位35_上电机反转	AT	%QX8134.4:BOOL;
	QX8134_5_工位35_下电机正转	AT	%QX8134.5:BOOL;
	QX8134_6_工位35_下电机反转	AT	%QX8134.6:BOOL;
	QX8134_7_工位35_预留	AT	%QX8134.7:BOOL;
	QX8135_0_工位36_指示灯_红	AT	%QX8135.0:BOOL;
	QX8135_1_工位36_指示灯_黄	AT	%QX8135.1:BOOL;
	QX8135_2_工位36_指示灯_绿	AT	%QX8135.2:BOOL;
	QX8135_3_工位36_上电机正转	AT	%QX8135.3:BOOL;
	QX8135_4_工位36_上电机反转	AT	%QX8135.4:BOOL;
	QX8135_5_工位36_下电机正转	AT	%QX8135.5:BOOL;
	QX8135_6_工位36_下电机反转	AT	%QX8135.6:BOOL;
	QX8135_7_工位36_40开关电源控制	AT	%QX8135.7:BOOL;
	QX8136_0_工位37_指示灯_红	AT	%QX8136.0:BOOL;
	QX8136_1_工位37_指示灯_黄	AT	%QX8136.1:BOOL;
	QX8136_2_工位37_指示灯_绿	AT	%QX8136.2:BOOL;
	QX8136_3_工位37_上电机正转	AT	%QX8136.3:BOOL;
	QX8136_4_工位37_上电机反转	AT	%QX8136.4:BOOL;
	QX8136_5_工位37_下电机正转	AT	%QX8136.5:BOOL;
	QX8136_6_工位37_下电机反转	AT	%QX8136.6:BOOL;
	QX8136_7_工位37_预留	AT	%QX8136.7:BOOL;
	QX8137_0_工位38_指示灯_红	AT	%QX8137.0:BOOL;
	QX8137_1_工位38_指示灯_黄	AT	%QX8137.1:BOOL;
	QX8137_2_工位38_指示灯_绿	AT	%QX8137.2:BOOL;
	QX8137_3_工位38_上电机正转	AT	%QX8137.3:BOOL;
	QX8137_4_工位38_上电机反转	AT	%QX8137.4:BOOL;
	QX8137_5_工位38_下电机正转	AT	%QX8137.5:BOOL;
	QX8137_6_工位38_下电机反转	AT	%QX8137.6:BOOL;
	QX8137_7_工位38_预留	AT	%QX8137.7:BOOL;
	QX8138_0_工位39_指示灯_红	AT	%QX8138.0:BOOL;
	QX8138_1_工位39_指示灯_黄	AT	%QX8138.1:BOOL;
	QX8138_2_工位39_指示灯_绿	AT	%QX8138.2:BOOL;
	QX8138_3_工位39_上电机正转	AT	%QX8138.3:BOOL;
	QX8138_4_工位39_上电机反转	AT	%QX8138.4:BOOL;
	QX8138_5_工位39_下电机正转	AT	%QX8138.5:BOOL;
	QX8138_6_工位39_下电机反转	AT	%QX8138.6:BOOL;
	QX8138_7_工位39_预留	AT	%QX8138.7:BOOL;
	QX8139_0_工位40_指示灯_红	AT	%QX8139.0:BOOL;
	QX8139_1_工位40_指示灯_黄	AT	%QX8139.1:BOOL;
	QX8139_2_工位40_指示灯_绿	AT	%QX8139.2:BOOL;
	QX8139_3_工位40_上电机正转	AT	%QX8139.3:BOOL;
	QX8139_4_工位40_上电机反转	AT	%QX8139.4:BOOL;
	QX8139_5_工位40_下电机正转	AT	%QX8139.5:BOOL;
	QX8139_6_工位40_下电机反转	AT	%QX8139.6:BOOL;
	QX8139_7_工位40_预留	AT	%QX8139.7:BOOL;
	QX8200_0_工位41_指示灯_红	AT	%QX8200.0:BOOL;
	QX8200_1_工位41_指示灯_黄	AT	%QX8200.1:BOOL;
	QX8200_2_工位41_指示灯_绿	AT	%QX8200.2:BOOL;
	QX8200_3_工位41_上电机正转	AT	%QX8200.3:BOOL;
	QX8200_4_工位41_上电机反转	AT	%QX8200.4:BOOL;
	QX8200_5_工位41_下电机正转	AT	%QX8200.5:BOOL;
	QX8200_6_工位41_下电机反转	AT	%QX8200.6:BOOL;
	QX8200_7_工位41_45开关电源控制	AT	%QX8200.7:BOOL;
	QX8201_0_工位42_指示灯_红	AT	%QX8201.0:BOOL;
	QX8201_1_工位42_指示灯_黄	AT	%QX8201.1:BOOL;
	QX8201_2_工位42_指示灯_绿	AT	%QX8201.2:BOOL;
	QX8201_3_工位42_上电机正转	AT	%QX8201.3:BOOL;
	QX8201_4_工位42_上电机反转	AT	%QX8201.4:BOOL;
	QX8201_5_工位42_下电机正转	AT	%QX8201.5:BOOL;
	QX8201_6_工位42_下电机反转	AT	%QX8201.6:BOOL;
	QX8201_7_工位42_预留	AT	%QX8201.7:BOOL;
	QX8202_0_工位43_指示灯_红	AT	%QX8202.0:BOOL;
	QX8202_1_工位43_指示灯_黄	AT	%QX8202.1:BOOL;
	QX8202_2_工位43_指示灯_绿	AT	%QX8202.2:BOOL;
	QX8202_3_工位43_上电机正转	AT	%QX8202.3:BOOL;
	QX8202_4_工位43_上电机反转	AT	%QX8202.4:BOOL;
	QX8202_5_工位43_下电机正转	AT	%QX8202.5:BOOL;
	QX8202_6_工位43_下电机反转	AT	%QX8202.6:BOOL;
	QX8202_7_工位43_预留	AT	%QX8202.7:BOOL;
	QX8203_0_工位44_指示灯_红	AT	%QX8203.0:BOOL;
	QX8203_1_工位44_指示灯_黄	AT	%QX8203.1:BOOL;
	QX8203_2_工位44_指示灯_绿	AT	%QX8203.2:BOOL;
	QX8203_3_工位44_上电机正转	AT	%QX8203.3:BOOL;
	QX8203_4_工位44_上电机反转	AT	%QX8203.4:BOOL;
	QX8203_5_工位44_下电机正转	AT	%QX8203.5:BOOL;
	QX8203_6_工位44_下电机反转	AT	%QX8203.6:BOOL;
	QX8203_7_工位44_预留	AT	%QX8203.7:BOOL;
	QX8204_0_工位45_指示灯_红	AT	%QX8204.0:BOOL;
	QX8204_1_工位45_指示灯_黄	AT	%QX8204.1:BOOL;
	QX8204_2_工位45_指示灯_绿	AT	%QX8204.2:BOOL;
	QX8204_3_工位45_上电机正转	AT	%QX8204.3:BOOL;
	QX8204_4_工位45_上电机反转	AT	%QX8204.4:BOOL;
	QX8204_5_工位45_下电机正转	AT	%QX8204.5:BOOL;
	QX8204_6_工位45_下电机反转	AT	%QX8204.6:BOOL;
	QX8204_7_工位45_预留	AT	%QX8204.7:BOOL;
	QX8205_0_工位46_指示灯_红	AT	%QX8205.0:BOOL;
	QX8205_1_工位46_指示灯_黄	AT	%QX8205.1:BOOL;
	QX8205_2_工位46_指示灯_绿	AT	%QX8205.2:BOOL;
	QX8205_3_工位46_上电机正转	AT	%QX8205.3:BOOL;
	QX8205_4_工位46_上电机反转	AT	%QX8205.4:BOOL;
	QX8205_5_工位46_下电机正转	AT	%QX8205.5:BOOL;
	QX8205_6_工位46_下电机反转	AT	%QX8205.6:BOOL;
	QX8205_7_工位46_50开关电源控制	AT	%QX8205.7:BOOL;
	QX8206_0_工位47_指示灯_红	AT	%QX8206.0:BOOL;
	QX8206_1_工位47_指示灯_黄	AT	%QX8206.1:BOOL;
	QX8206_2_工位47_指示灯_绿	AT	%QX8206.2:BOOL;
	QX8206_3_工位47_上电机正转	AT	%QX8206.3:BOOL;
	QX8206_4_工位47_上电机反转	AT	%QX8206.4:BOOL;
	QX8206_5_工位47_下电机正转	AT	%QX8206.5:BOOL;
	QX8206_6_工位47_下电机反转	AT	%QX8206.6:BOOL;
	QX8206_7_工位47_预留	AT	%QX8206.7:BOOL;
	QX8207_0_工位48_指示灯_红	AT	%QX8207.0:BOOL;
	QX8207_1_工位48_指示灯_黄	AT	%QX8207.1:BOOL;
	QX8207_2_工位48_指示灯_绿	AT	%QX8207.2:BOOL;
	QX8207_3_工位48_上电机正转	AT	%QX8207.3:BOOL;
	QX8207_4_工位48_上电机反转	AT	%QX8207.4:BOOL;
	QX8207_5_工位48_下电机正转	AT	%QX8207.5:BOOL;
	QX8207_6_工位48_下电机反转	AT	%QX8207.6:BOOL;
	QX8207_7_工位48_预留	AT	%QX8207.7:BOOL;
	QX8208_0_工位49_指示灯_红	AT	%QX8208.0:BOOL;
	QX8208_1_工位49_指示灯_黄	AT	%QX8208.1:BOOL;
	QX8208_2_工位49_指示灯_绿	AT	%QX8208.2:BOOL;
	QX8208_3_工位49_上电机正转	AT	%QX8208.3:BOOL;
	QX8208_4_工位49_上电机反转	AT	%QX8208.4:BOOL;
	QX8208_5_工位49_下电机正转	AT	%QX8208.5:BOOL;
	QX8208_6_工位49_下电机反转	AT	%QX8208.6:BOOL;
	QX8208_7_工位49_预留	AT	%QX8208.7:BOOL;
	QX8209_0_工位50_指示灯_红	AT	%QX8209.0:BOOL;
	QX8209_1_工位50_指示灯_黄	AT	%QX8209.1:BOOL;
	QX8209_2_工位50_指示灯_绿	AT	%QX8209.2:BOOL;
	QX8209_3_工位50_上电机正转	AT	%QX8209.3:BOOL;
	QX8209_4_工位50_上电机反转	AT	%QX8209.4:BOOL;
	QX8209_5_工位50_下电机正转	AT	%QX8209.5:BOOL;
	QX8209_6_工位50_下电机反转	AT	%QX8209.6:BOOL;
	QX8209_7_工位50_预留	AT	%QX8209.7:BOOL;
	QX8210_0_工位51_指示灯_红	AT	%QX8210.0:BOOL;
	QX8210_1_工位51_指示灯_黄	AT	%QX8210.1:BOOL;
	QX8210_2_工位51_指示灯_绿	AT	%QX8210.2:BOOL;
	QX8210_3_工位51_上电机正转	AT	%QX8210.3:BOOL;
	QX8210_4_工位51_上电机反转	AT	%QX8210.4:BOOL;
	QX8210_5_工位51_下电机正转	AT	%QX8210.5:BOOL;
	QX8210_6_工位51_下电机反转	AT	%QX8210.6:BOOL;
	QX8210_7_工位51_55开关电源控制	AT	%QX8210.7:BOOL;
	QX8211_0_工位52_指示灯_红	AT	%QX8211.0:BOOL;
	QX8211_1_工位52_指示灯_黄	AT	%QX8211.1:BOOL;
	QX8211_2_工位52_指示灯_绿	AT	%QX8211.2:BOOL;
	QX8211_3_工位52_上电机正转	AT	%QX8211.3:BOOL;
	QX8211_4_工位52_上电机反转	AT	%QX8211.4:BOOL;
	QX8211_5_工位52_下电机正转	AT	%QX8211.5:BOOL;
	QX8211_6_工位52_下电机反转	AT	%QX8211.6:BOOL;
	QX8211_7_工位52_预留	AT	%QX8211.7:BOOL;
	QX8212_0_工位53_指示灯_红	AT	%QX8212.0:BOOL;
	QX8212_1_工位53_指示灯_黄	AT	%QX8212.1:BOOL;
	QX8212_2_工位53_指示灯_绿	AT	%QX8212.2:BOOL;
	QX8212_3_工位53_上电机正转	AT	%QX8212.3:BOOL;
	QX8212_4_工位53_上电机反转	AT	%QX8212.4:BOOL;
	QX8212_5_工位53_下电机正转	AT	%QX8212.5:BOOL;
	QX8212_6_工位53_下电机反转	AT	%QX8212.6:BOOL;
	QX8212_7_工位53_预留	AT	%QX8212.7:BOOL;
	QX8213_0_工位54_指示灯_红	AT	%QX8213.0:BOOL;
	QX8213_1_工位54_指示灯_黄	AT	%QX8213.1:BOOL;
	QX8213_2_工位54_指示灯_绿	AT	%QX8213.2:BOOL;
	QX8213_3_工位54_上电机正转	AT	%QX8213.3:BOOL;
	QX8213_4_工位54_上电机反转	AT	%QX8213.4:BOOL;
	QX8213_5_工位54_下电机正转	AT	%QX8213.5:BOOL;
	QX8213_6_工位54_下电机反转	AT	%QX8213.6:BOOL;
	QX8213_7_工位54_预留	AT	%QX8213.7:BOOL;
	QX8214_0_工位55_指示灯_红	AT	%QX8214.0:BOOL;
	QX8214_1_工位55_指示灯_黄	AT	%QX8214.1:BOOL;
	QX8214_2_工位55_指示灯_绿	AT	%QX8214.2:BOOL;
	QX8214_3_工位55_上电机正转	AT	%QX8214.3:BOOL;
	QX8214_4_工位55_上电机反转	AT	%QX8214.4:BOOL;
	QX8214_5_工位55_下电机正转	AT	%QX8214.5:BOOL;
	QX8214_6_工位55_下电机反转	AT	%QX8214.6:BOOL;
	QX8214_7_工位55_预留	AT	%QX8214.7:BOOL;
	QX8215_0_工位56_指示灯_红	AT	%QX8215.0:BOOL;
	QX8215_1_工位56_指示灯_黄	AT	%QX8215.1:BOOL;
	QX8215_2_工位56_指示灯_绿	AT	%QX8215.2:BOOL;
	QX8215_3_工位56_上电机正转	AT	%QX8215.3:BOOL;
	QX8215_4_工位56_上电机反转	AT	%QX8215.4:BOOL;
	QX8215_5_工位56_下电机正转	AT	%QX8215.5:BOOL;
	QX8215_6_工位56_下电机反转	AT	%QX8215.6:BOOL;
	QX8215_7_工位56_60开关电源控制	AT	%QX8215.7:BOOL;
	QX8216_0_工位57_指示灯_红	AT	%QX8216.0:BOOL;
	QX8216_1_工位57_指示灯_黄	AT	%QX8216.1:BOOL;
	QX8216_2_工位57_指示灯_绿	AT	%QX8216.2:BOOL;
	QX8216_3_工位57_上电机正转	AT	%QX8216.3:BOOL;
	QX8216_4_工位57_上电机反转	AT	%QX8216.4:BOOL;
	QX8216_5_工位57_下电机正转	AT	%QX8216.5:BOOL;
	QX8216_6_工位57_下电机反转	AT	%QX8216.6:BOOL;
	QX8216_7_工位57_预留	AT	%QX8216.7:BOOL;
	QX8217_0_工位58_指示灯_红	AT	%QX8217.0:BOOL;
	QX8217_1_工位58_指示灯_黄	AT	%QX8217.1:BOOL;
	QX8217_2_工位58_指示灯_绿	AT	%QX8217.2:BOOL;
	QX8217_3_工位58_上电机正转	AT	%QX8217.3:BOOL;
	QX8217_4_工位58_上电机反转	AT	%QX8217.4:BOOL;
	QX8217_5_工位58_下电机正转	AT	%QX8217.5:BOOL;
	QX8217_6_工位58_下电机反转	AT	%QX8217.6:BOOL;
	QX8217_7_工位58_预留	AT	%QX8217.7:BOOL;
	QX8218_0_工位59_指示灯_红	AT	%QX8218.0:BOOL;
	QX8218_1_工位59_指示灯_黄	AT	%QX8218.1:BOOL;
	QX8218_2_工位59_指示灯_绿	AT	%QX8218.2:BOOL;
	QX8218_3_工位59_上电机正转	AT	%QX8218.3:BOOL;
	QX8218_4_工位59_上电机反转	AT	%QX8218.4:BOOL;
	QX8218_5_工位59_下电机正转	AT	%QX8218.5:BOOL;
	QX8218_6_工位59_下电机反转	AT	%QX8218.6:BOOL;
	QX8218_7_工位59_预留	AT	%QX8218.7:BOOL;
	QX8219_0_工位60_指示灯_红	AT	%QX8219.0:BOOL;
	QX8219_1_工位60_指示灯_黄	AT	%QX8219.1:BOOL;
	QX8219_2_工位60_指示灯_绿	AT	%QX8219.2:BOOL;
	QX8219_3_工位60_上电机正转	AT	%QX8219.3:BOOL;
	QX8219_4_工位60_上电机反转	AT	%QX8219.4:BOOL;
	QX8219_5_工位60_下电机正转	AT	%QX8219.5:BOOL;
	QX8219_6_工位60_下电机反转	AT	%QX8219.6:BOOL;
	QX8219_7_工位60_预留	AT	%QX8219.7:BOOL;
	QX8220_0_工位61_指示灯_红	AT	%QX8220.0:BOOL;
	QX8220_1_工位61_指示灯_黄	AT	%QX8220.1:BOOL;
	QX8220_2_工位61_指示灯_绿	AT	%QX8220.2:BOOL;
	QX8220_3_工位61_上电机正转	AT	%QX8220.3:BOOL;
	QX8220_4_工位61_上电机反转	AT	%QX8220.4:BOOL;
	QX8220_5_工位61_下电机正转	AT	%QX8220.5:BOOL;
	QX8220_6_工位61_下电机反转	AT	%QX8220.6:BOOL;
	QX8220_7_工位61_65开关电源控制	AT	%QX8220.7:BOOL;
	QX8221_0_工位62_指示灯_红	AT	%QX8221.0:BOOL;
	QX8221_1_工位62_指示灯_黄	AT	%QX8221.1:BOOL;
	QX8221_2_工位62_指示灯_绿	AT	%QX8221.2:BOOL;
	QX8221_3_工位62_上电机正转	AT	%QX8221.3:BOOL;
	QX8221_4_工位62_上电机反转	AT	%QX8221.4:BOOL;
	QX8221_5_工位62_下电机正转	AT	%QX8221.5:BOOL;
	QX8221_6_工位62_下电机反转	AT	%QX8221.6:BOOL;
	QX8221_7_工位62_预留	AT	%QX8221.7:BOOL;
	QX8222_0_工位63_指示灯_红	AT	%QX8222.0:BOOL;
	QX8222_1_工位63_指示灯_黄	AT	%QX8222.1:BOOL;
	QX8222_2_工位63_指示灯_绿	AT	%QX8222.2:BOOL;
	QX8222_3_工位63_上电机正转	AT	%QX8222.3:BOOL;
	QX8222_4_工位63_上电机反转	AT	%QX8222.4:BOOL;
	QX8222_5_工位63_下电机正转	AT	%QX8222.5:BOOL;
	QX8222_6_工位63_下电机反转	AT	%QX8222.6:BOOL;
	QX8222_7_工位63_预留	AT	%QX8222.7:BOOL;
	QX8223_0_工位64_指示灯_红	AT	%QX8223.0:BOOL;
	QX8223_1_工位64_指示灯_黄	AT	%QX8223.1:BOOL;
	QX8223_2_工位64_指示灯_绿	AT	%QX8223.2:BOOL;
	QX8223_3_工位64_上电机正转	AT	%QX8223.3:BOOL;
	QX8223_4_工位64_上电机反转	AT	%QX8223.4:BOOL;
	QX8223_5_工位64_下电机正转	AT	%QX8223.5:BOOL;
	QX8223_6_工位64_下电机反转	AT	%QX8223.6:BOOL;
	QX8223_7_工位64_预留	AT	%QX8223.7:BOOL;
	QX8224_0_工位65_指示灯_红	AT	%QX8224.0:BOOL;
	QX8224_1_工位65_指示灯_黄	AT	%QX8224.1:BOOL;
	QX8224_2_工位65_指示灯_绿	AT	%QX8224.2:BOOL;
	QX8224_3_工位65_上电机正转	AT	%QX8224.3:BOOL;
	QX8224_4_工位65_上电机反转	AT	%QX8224.4:BOOL;
	QX8224_5_工位65_下电机正转	AT	%QX8224.5:BOOL;
	QX8224_6_工位65_下电机反转	AT	%QX8224.6:BOOL;
	QX8224_7_工位65_预留	AT	%QX8224.7:BOOL;
	QX8225_0_工位66_指示灯_红	AT	%QX8225.0:BOOL;
	QX8225_1_工位66_指示灯_黄	AT	%QX8225.1:BOOL;
	QX8225_2_工位66_指示灯_绿	AT	%QX8225.2:BOOL;
	QX8225_3_工位66_上电机正转	AT	%QX8225.3:BOOL;
	QX8225_4_工位66_上电机反转	AT	%QX8225.4:BOOL;
	QX8225_5_工位66_下电机正转	AT	%QX8225.5:BOOL;
	QX8225_6_工位66_下电机反转	AT	%QX8225.6:BOOL;
	QX8225_7_工位66_70开关电源控制	AT	%QX8225.7:BOOL;
	QX8226_0_工位67_指示灯_红	AT	%QX8226.0:BOOL;
	QX8226_1_工位67_指示灯_黄	AT	%QX8226.1:BOOL;
	QX8226_2_工位67_指示灯_绿	AT	%QX8226.2:BOOL;
	QX8226_3_工位67_上电机正转	AT	%QX8226.3:BOOL;
	QX8226_4_工位67_上电机反转	AT	%QX8226.4:BOOL;
	QX8226_5_工位67_下电机正转	AT	%QX8226.5:BOOL;
	QX8226_6_工位67_下电机反转	AT	%QX8226.6:BOOL;
	QX8226_7_工位67_预留	AT	%QX8226.7:BOOL;
	QX8227_0_工位68_指示灯_红	AT	%QX8227.0:BOOL;
	QX8227_1_工位68_指示灯_黄	AT	%QX8227.1:BOOL;
	QX8227_2_工位68_指示灯_绿	AT	%QX8227.2:BOOL;
	QX8227_3_工位68_上电机正转	AT	%QX8227.3:BOOL;
	QX8227_4_工位68_上电机反转	AT	%QX8227.4:BOOL;
	QX8227_5_工位68_下电机正转	AT	%QX8227.5:BOOL;
	QX8227_6_工位68_下电机反转	AT	%QX8227.6:BOOL;
	QX8227_7_工位68_预留	AT	%QX8227.7:BOOL;
	QX8228_0_工位69_指示灯_红	AT	%QX8228.0:BOOL;
	QX8228_1_工位69_指示灯_黄	AT	%QX8228.1:BOOL;
	QX8228_2_工位69_指示灯_绿	AT	%QX8228.2:BOOL;
	QX8228_3_工位69_上电机正转	AT	%QX8228.3:BOOL;
	QX8228_4_工位69_上电机反转	AT	%QX8228.4:BOOL;
	QX8228_5_工位69_下电机正转	AT	%QX8228.5:BOOL;
	QX8228_6_工位69_下电机反转	AT	%QX8228.6:BOOL;
	QX8228_7_工位69_预留	AT	%QX8228.7:BOOL;
	QX8229_0_工位70_指示灯_红	AT	%QX8229.0:BOOL;
	QX8229_1_工位70_指示灯_黄	AT	%QX8229.1:BOOL;
	QX8229_2_工位70_指示灯_绿	AT	%QX8229.2:BOOL;
	QX8229_3_工位70_上电机正转	AT	%QX8229.3:BOOL;
	QX8229_4_工位70_上电机反转	AT	%QX8229.4:BOOL;
	QX8229_5_工位70_下电机正转	AT	%QX8229.5:BOOL;
	QX8229_6_工位70_下电机反转	AT	%QX8229.6:BOOL;
	QX8229_7_工位70_预留	AT	%QX8229.7:BOOL;
	QX8230_0_工位71_指示灯_红	AT	%QX8230.0:BOOL;
	QX8230_1_工位71_指示灯_黄	AT	%QX8230.1:BOOL;
	QX8230_2_工位71_指示灯_绿	AT	%QX8230.2:BOOL;
	QX8230_3_工位71_上电机正转	AT	%QX8230.3:BOOL;
	QX8230_4_工位71_上电机反转	AT	%QX8230.4:BOOL;
	QX8230_5_工位71_下电机正转	AT	%QX8230.5:BOOL;
	QX8230_6_工位71_下电机反转	AT	%QX8230.6:BOOL;
	QX8230_7_工位71_75开关电源控制	AT	%QX8230.7:BOOL;
	QX8231_0_工位72_指示灯_红	AT	%QX8231.0:BOOL;
	QX8231_1_工位72_指示灯_黄	AT	%QX8231.1:BOOL;
	QX8231_2_工位72_指示灯_绿	AT	%QX8231.2:BOOL;
	QX8231_3_工位72_上电机正转	AT	%QX8231.3:BOOL;
	QX8231_4_工位72_上电机反转	AT	%QX8231.4:BOOL;
	QX8231_5_工位72_下电机正转	AT	%QX8231.5:BOOL;
	QX8231_6_工位72_下电机反转	AT	%QX8231.6:BOOL;
	QX8231_7_工位72_预留	AT	%QX8231.7:BOOL;
	QX8232_0_工位73_指示灯_红	AT	%QX8232.0:BOOL;
	QX8232_1_工位73_指示灯_黄	AT	%QX8232.1:BOOL;
	QX8232_2_工位73_指示灯_绿	AT	%QX8232.2:BOOL;
	QX8232_3_工位73_上电机正转	AT	%QX8232.3:BOOL;
	QX8232_4_工位73_上电机反转	AT	%QX8232.4:BOOL;
	QX8232_5_工位73_下电机正转	AT	%QX8232.5:BOOL;
	QX8232_6_工位73_下电机反转	AT	%QX8232.6:BOOL;
	QX8232_7_工位73_预留	AT	%QX8232.7:BOOL;
	QX8233_0_工位74_指示灯_红	AT	%QX8233.0:BOOL;
	QX8233_1_工位74_指示灯_黄	AT	%QX8233.1:BOOL;
	QX8233_2_工位74_指示灯_绿	AT	%QX8233.2:BOOL;
	QX8233_3_工位74_上电机正转	AT	%QX8233.3:BOOL;
	QX8233_4_工位74_上电机反转	AT	%QX8233.4:BOOL;
	QX8233_5_工位74_下电机正转	AT	%QX8233.5:BOOL;
	QX8233_6_工位74_下电机反转	AT	%QX8233.6:BOOL;
	QX8233_7_工位74_预留	AT	%QX8233.7:BOOL;
	QX8234_0_工位75_指示灯_红	AT	%QX8234.0:BOOL;
	QX8234_1_工位75_指示灯_黄	AT	%QX8234.1:BOOL;
	QX8234_2_工位75_指示灯_绿	AT	%QX8234.2:BOOL;
	QX8234_3_工位75_上电机正转	AT	%QX8234.3:BOOL;
	QX8234_4_工位75_上电机反转	AT	%QX8234.4:BOOL;
	QX8234_5_工位75_下电机正转	AT	%QX8234.5:BOOL;
	QX8234_6_工位75_下电机反转	AT	%QX8234.6:BOOL;
	QX8234_7_工位75_预留	AT	%QX8234.7:BOOL;
	QX8235_0_工位76_指示灯_红	AT	%QX8235.0:BOOL;
	QX8235_1_工位76_指示灯_黄	AT	%QX8235.1:BOOL;
	QX8235_2_工位76_指示灯_绿	AT	%QX8235.2:BOOL;
	QX8235_3_工位76_上电机正转	AT	%QX8235.3:BOOL;
	QX8235_4_工位76_上电机反转	AT	%QX8235.4:BOOL;
	QX8235_5_工位76_下电机正转	AT	%QX8235.5:BOOL;
	QX8235_6_工位76_下电机反转	AT	%QX8235.6:BOOL;
	QX8235_7_工位76_80开关电源控制	AT	%QX8235.7:BOOL;
	QX8236_0_工位77_指示灯_红	AT	%QX8236.0:BOOL;
	QX8236_1_工位77_指示灯_黄	AT	%QX8236.1:BOOL;
	QX8236_2_工位77_指示灯_绿	AT	%QX8236.2:BOOL;
	QX8236_3_工位77_上电机正转	AT	%QX8236.3:BOOL;
	QX8236_4_工位77_上电机反转	AT	%QX8236.4:BOOL;
	QX8236_5_工位77_下电机正转	AT	%QX8236.5:BOOL;
	QX8236_6_工位77_下电机反转	AT	%QX8236.6:BOOL;
	QX8236_7_工位77_预留	AT	%QX8236.7:BOOL;
	QX8237_0_工位78_指示灯_红	AT	%QX8237.0:BOOL;
	QX8237_1_工位78_指示灯_黄	AT	%QX8237.1:BOOL;
	QX8237_2_工位78_指示灯_绿	AT	%QX8237.2:BOOL;
	QX8237_3_工位78_上电机正转	AT	%QX8237.3:BOOL;
	QX8237_4_工位78_上电机反转	AT	%QX8237.4:BOOL;
	QX8237_5_工位78_下电机正转	AT	%QX8237.5:BOOL;
	QX8237_6_工位78_下电机反转	AT	%QX8237.6:BOOL;
	QX8237_7_工位78_预留	AT	%QX8237.7:BOOL;
	QX8238_0_工位79_指示灯_红	AT	%QX8238.0:BOOL;
	QX8238_1_工位79_指示灯_黄	AT	%QX8238.1:BOOL;
	QX8238_2_工位79_指示灯_绿	AT	%QX8238.2:BOOL;
	QX8238_3_工位79_上电机正转	AT	%QX8238.3:BOOL;
	QX8238_4_工位79_上电机反转	AT	%QX8238.4:BOOL;
	QX8238_5_工位79_下电机正转	AT	%QX8238.5:BOOL;
	QX8238_6_工位79_下电机反转	AT	%QX8238.6:BOOL;
	QX8238_7_工位79_预留	AT	%QX8238.7:BOOL;
	QX8239_0_工位80_指示灯_红	AT	%QX8239.0:BOOL;
	QX8239_1_工位80_指示灯_黄	AT	%QX8239.1:BOOL;
	QX8239_2_工位80_指示灯_绿	AT	%QX8239.2:BOOL;
	QX8239_3_工位80_上电机正转	AT	%QX8239.3:BOOL;
	QX8239_4_工位80_上电机反转	AT	%QX8239.4:BOOL;
	QX8239_5_工位80_下电机正转	AT	%QX8239.5:BOOL;
	QX8239_6_工位80_下电机反转	AT	%QX8239.6:BOOL;
	QX8239_7_工位80_预留	AT	%QX8239.7:BOOL;
	QX8300_0_测试1_产品侧边定位气缸CY01_伸出	AT	%QX8300.0:BOOL;
	QX8300_1_测试1_产品侧边定位气缸CY01_缩回	AT	%QX8300.1:BOOL;
	QX8300_2_测试1_产品固定气缸CY02_锁紧	AT	%QX8300.2:BOOL;
	QX8300_3_测试1_产品固定气缸CY02_松开	AT	%QX8300.3:BOOL;
	QX8300_4	AT	%QX8300.4:BOOL;
	QX8300_5	AT	%QX8300.5:BOOL;
	QX8300_6_测试1_产品封堵A上下气缸CY03_上升	AT	%QX8300.6:BOOL;
	QX8300_7_测试1_产品封堵A上下气缸CY03_下降	AT	%QX8300.7:BOOL;
	QX8301_0_测试1_产品封堵A侧推气缸CY04_伸出	AT	%QX8301.0:BOOL;
	QX8301_1_测试1_产品封堵A侧推气缸CY04_缩回	AT	%QX8301.1:BOOL;
	QX8301_2_测试1_产品封堵B上下气缸CY05_上升	AT	%QX8301.2:BOOL;
	QX8301_3_测试1_产品封堵B上下气缸CY05_下降	AT	%QX8301.3:BOOL;
	QX8301_4_测试1_驱动齿轮气缸CY06_伸出	AT	%QX8301.4:BOOL;
	QX8301_5_测试1_驱动齿轮气缸CY06_缩回	AT	%QX8301.5:BOOL;
	QX8301_6_测试1_固定夹爪气缸CY07_夹紧	AT	%QX8301.6:BOOL;
	QX8301_7_测试1_固定夹爪气缸CY07_缩回	AT	%QX8301.7:BOOL;
	QX8302_0_测试1_插管测试气缸CY08_上升	AT	%QX8302.0:BOOL;
	QX8302_1_测试1_插管测试气缸CY08_下降	AT	%QX8302.1:BOOL;
	QX8302_2_测试1_拔管解扣气缸CY09_上升	AT	%QX8302.2:BOOL;
	QX8302_3_测试1_拔管解扣气缸CY09_下降	AT	%QX8302.3:BOOL;
	QX8302_4_缓存NG1_侧边定位气缸CY10_伸出	AT	%QX8302.4:BOOL;
	QX8302_5_缓存NG1_侧边定位气缸CY10_缩回	AT	%QX8302.5:BOOL;
	QX8302_6	AT	%QX8302.6:BOOL;
	QX8302_7	AT	%QX8302.7:BOOL;
	QX8303_0	AT	%QX8303.0:BOOL;
	QX8303_1	AT	%QX8303.1:BOOL;
	QX8303_2	AT	%QX8303.2:BOOL;
	QX8303_3_测试1_双手启动按钮_左指示灯	AT	%QX8303.3:BOOL;
	QX8303_4_测试1_双手启动按钮_右指示灯	AT	%QX8303.4:BOOL;
	QX8303_5	AT	%QX8303.5:BOOL;
	QX8303_6	AT	%QX8303.6:BOOL;
	QX8303_7	AT	%QX8303.7:BOOL;
	QX8304_0_测试2_产品侧边定位气缸CY11_伸出	AT	%QX8304.0:BOOL;
	QX8304_1_测试2_产品侧边定位气缸CY11_缩回	AT	%QX8304.1:BOOL;
	QX8304_2_测试2_产品固定气缸CY12_锁紧	AT	%QX8304.2:BOOL;
	QX8304_3_测试2_产品固定气缸CY12_松开	AT	%QX8304.3:BOOL;
	QX8304_4	AT	%QX8304.4:BOOL;
	QX8304_5	AT	%QX8304.5:BOOL;
	QX8304_6_测试2_产品封堵A上下气缸CY13_上升	AT	%QX8304.6:BOOL;
	QX8304_7_测试2_产品封堵A上下气缸CY13_下降	AT	%QX8304.7:BOOL;
	QX8305_0_测试2_产品封堵A侧推气缸CY14_伸出	AT	%QX8305.0:BOOL;
	QX8305_1_测试2_产品封堵A侧推气缸CY14_缩回	AT	%QX8305.1:BOOL;
	QX8305_2_测试2_产品封堵B上下气缸CY15_上升	AT	%QX8305.2:BOOL;
	QX8305_3_测试2_产品封堵B上下气缸CY15_下降	AT	%QX8305.3:BOOL;
	QX8305_4_测试2_驱动齿轮气缸CY16_伸出	AT	%QX8305.4:BOOL;
	QX8305_5_测试2_驱动齿轮气缸CY16_缩回	AT	%QX8305.5:BOOL;
	QX8305_6_测试2_固定夹爪气缸CY17_夹紧	AT	%QX8305.6:BOOL;
	QX8305_7_测试2_固定夹爪气缸CY17_缩回	AT	%QX8305.7:BOOL;
	QX8306_0_测试2_插管测试气缸CY18_上升	AT	%QX8306.0:BOOL;
	QX8306_1_测试2_插管测试气缸CY18_下降	AT	%QX8306.1:BOOL;
	QX8306_2_测试2_拔管解扣气缸CY19_上升	AT	%QX8306.2:BOOL;
	QX8306_3_测试2_拔管解扣气缸CY19_下降	AT	%QX8306.3:BOOL;
	QX8306_4_缓存NG2_侧边定位气缸CY20_伸出	AT	%QX8306.4:BOOL;
	QX8306_5_缓存NG2_侧边定位气缸CY20_缩回	AT	%QX8306.5:BOOL;
	QX8306_6	AT	%QX8306.6:BOOL;
	QX8306_7	AT	%QX8306.7:BOOL;
	QX8307_0	AT	%QX8307.0:BOOL;
	QX8307_1	AT	%QX8307.1:BOOL;
	QX8307_2	AT	%QX8307.2:BOOL;
	QX8307_3_测试2_双手启动按钮_左指示灯	AT	%QX8307.3:BOOL;
	QX8307_4_测试2_双手启动按钮_右指示灯	AT	%QX8307.4:BOOL;
	QX8307_5	AT	%QX8307.5:BOOL;
	QX8307_6	AT	%QX8307.6:BOOL;
	QX8307_7	AT	%QX8307.7:BOOL;
	QX8400_0_测试3_产品侧边定位气缸CY21_伸出	AT	%QX8400.0:BOOL;
	QX8400_1_测试3_产品侧边定位气缸CY21_缩回	AT	%QX8400.1:BOOL;
	QX8400_2_测试3_产品固定气缸CY22_锁紧	AT	%QX8400.2:BOOL;
	QX8400_3_测试3_产品固定气缸CY22_松开	AT	%QX8400.3:BOOL;
	QX8400_4	AT	%QX8400.4:BOOL;
	QX8400_5	AT	%QX8400.5:BOOL;
	QX8400_6_测试3_产品封堵A上下气缸CY23_上升	AT	%QX8400.6:BOOL;
	QX8400_7_测试3_产品封堵A上下气缸CY23_下降	AT	%QX8400.7:BOOL;
	QX8401_0_测试3_产品封堵A侧推气缸CY24_伸出	AT	%QX8401.0:BOOL;
	QX8401_1_测试3_产品封堵A侧推气缸CY24_缩回	AT	%QX8401.1:BOOL;
	QX8401_2_测试3_产品封堵B上下气缸CY25_上升	AT	%QX8401.2:BOOL;
	QX8401_3_测试3_产品封堵B上下气缸CY25_下降	AT	%QX8401.3:BOOL;
	QX8401_4_测试3_驱动齿轮气缸CY26_伸出	AT	%QX8401.4:BOOL;
	QX8401_5_测试3_驱动齿轮气缸CY26_缩回	AT	%QX8401.5:BOOL;
	QX8401_6_测试3_固定夹爪气缸CY27_夹紧	AT	%QX8401.6:BOOL;
	QX8401_7_测试3_固定夹爪气缸CY27_缩回	AT	%QX8401.7:BOOL;
	QX8402_0_测试3_插管测试气缸CY28_上升	AT	%QX8402.0:BOOL;
	QX8402_1_测试3_插管测试气缸CY28_下降	AT	%QX8402.1:BOOL;
	QX8402_2_测试3_拔管解扣气缸CY29_上升	AT	%QX8402.2:BOOL;
	QX8402_3_测试3_拔管解扣气缸CY29_下降	AT	%QX8402.3:BOOL;
	QX8402_4_缓存NG3_侧边定位气缸CY30_伸出	AT	%QX8402.4:BOOL;
	QX8402_5_缓存NG3_侧边定位气缸CY30_缩回	AT	%QX8402.5:BOOL;
	QX8402_6	AT	%QX8402.6:BOOL;
	QX8402_7	AT	%QX8402.7:BOOL;
	QX8403_0	AT	%QX8403.0:BOOL;
	QX8403_1	AT	%QX8403.1:BOOL;
	QX8403_2	AT	%QX8403.2:BOOL;
	QX8403_3_测试3_双手启动按钮_左指示灯	AT	%QX8403.3:BOOL;
	QX8403_4_测试3_双手启动按钮_右指示灯	AT	%QX8403.4:BOOL;
	QX8403_5	AT	%QX8403.5:BOOL;
	QX8403_6	AT	%QX8403.6:BOOL;
	QX8403_7	AT	%QX8403.7:BOOL;
	QX8404_0_测试4_产品侧边定位气缸CY31_伸出	AT	%QX8404.0:BOOL;
	QX8404_1_测试4_产品侧边定位气缸CY31_缩回	AT	%QX8404.1:BOOL;
	QX8404_2_测试4_产品固定气缸CY32_锁紧	AT	%QX8404.2:BOOL;
	QX8404_3_测试4_产品固定气缸CY32_松开	AT	%QX8404.3:BOOL;
	QX8404_4	AT	%QX8404.4:BOOL;
	QX8404_5	AT	%QX8404.5:BOOL;
	QX8404_6_测试4_产品封堵A上下气缸CY33_上升	AT	%QX8404.6:BOOL;
	QX8404_7_测试4_产品封堵A上下气缸CY33_下降	AT	%QX8404.7:BOOL;
	QX8405_0_测试4_产品封堵A侧推气缸CY34_伸出	AT	%QX8405.0:BOOL;
	QX8405_1_测试4_产品封堵A侧推气缸CY34_缩回	AT	%QX8405.1:BOOL;
	QX8405_2_测试4_产品封堵B上下气缸CY35_上升	AT	%QX8405.2:BOOL;
	QX8405_3_测试4_产品封堵B上下气缸CY35_下降	AT	%QX8405.3:BOOL;
	QX8405_4_测试4_驱动齿轮气缸CY36_伸出	AT	%QX8405.4:BOOL;
	QX8405_5_测试4_驱动齿轮气缸CY36_缩回	AT	%QX8405.5:BOOL;
	QX8405_6_测试4_固定夹爪气缸CY37_夹紧	AT	%QX8405.6:BOOL;
	QX8405_7_测试4_固定夹爪气缸CY37_缩回	AT	%QX8405.7:BOOL;
	QX8406_0_测试4_插管测试气缸CY38_上升	AT	%QX8406.0:BOOL;
	QX8406_1_测试4_插管测试气缸CY38_下降	AT	%QX8406.1:BOOL;
	QX8406_2_测试4_拔管解扣气缸CY39_上升	AT	%QX8406.2:BOOL;
	QX8406_3_测试4_拔管解扣气缸CY39_下降	AT	%QX8406.3:BOOL;
	QX8406_4_缓存NG4_侧边定位气缸CY40_伸出	AT	%QX8406.4:BOOL;
	QX8406_5_缓存NG4_侧边定位气缸CY40_缩回	AT	%QX8406.5:BOOL;
	QX8406_6	AT	%QX8406.6:BOOL;
	QX8406_7	AT	%QX8406.7:BOOL;
	QX8407_0	AT	%QX8407.0:BOOL;
	QX8407_1	AT	%QX8407.1:BOOL;
	QX8407_2	AT	%QX8407.2:BOOL;
	QX8407_3_测试4_双手启动按钮_左指示灯	AT	%QX8407.3:BOOL;
	QX8407_4_测试4_双手启动按钮_右指示灯	AT	%QX8407.4:BOOL;
	QX8407_5	AT	%QX8407.5:BOOL;
	QX8407_6	AT	%QX8407.6:BOOL;
	QX8407_7	AT	%QX8407.7:BOOL;
	QX8500_0_上料机械手夹爪CY41_夹紧	AT	%QX8500.0:BOOL;
	QX8500_1_上料机械手夹爪CY41_打开	AT	%QX8500.1:BOOL;
	QX8500_2	AT	%QX8500.2:BOOL;
	QX8500_3	AT	%QX8500.3:BOOL;
	QX8500_4	AT	%QX8500.4:BOOL;
	QX8500_5	AT	%QX8500.5:BOOL;
	QX8500_6	AT	%QX8500.6:BOOL;
	QX8500_7	AT	%QX8500.7:BOOL;
	QX8501_0	AT	%QX8501.0:BOOL;
	QX8501_1	AT	%QX8501.1:BOOL;
	QX8501_2	AT	%QX8501.2:BOOL;
	QX8501_3	AT	%QX8501.3:BOOL;
	QX8501_4	AT	%QX8501.4:BOOL;
	QX8501_5	AT	%QX8501.5:BOOL;
	QX8501_6	AT	%QX8501.6:BOOL;
	QX8501_7	AT	%QX8501.7:BOOL;
	QX8600_0_码垛机械手夹爪CY45_夹紧	AT	%QX8600.0:BOOL;
	QX8600_1_码垛机械手夹爪CY45_打开	AT	%QX8600.1:BOOL;
	QX8600_2_码垛机械手隔板真空吸Vac01_吸真空	AT	%QX8600.2:BOOL;
	QX8600_3_码垛机械手隔板真空吸Vac01_破真空	AT	%QX8600.3:BOOL;
	QX8600_4	AT	%QX8600.4:BOOL;
	QX8600_5	AT	%QX8600.5:BOOL;
	QX8600_6	AT	%QX8600.6:BOOL;
	QX8600_7	AT	%QX8600.7:BOOL;
	QX8601_0	AT	%QX8601.0:BOOL;
	QX8601_1	AT	%QX8601.1:BOOL;
	QX8601_2	AT	%QX8601.2:BOOL;
	QX8601_3	AT	%QX8601.3:BOOL;
	QX8601_4	AT	%QX8601.4:BOOL;
	QX8601_5	AT	%QX8601.5:BOOL;
	QX8601_6	AT	%QX8601.6:BOOL;
	QX8601_7	AT	%QX8601.7:BOOL;
	QX8700_0_皮带线启动	AT	%QX8700.0:BOOL;
	QX8700_1	AT	%QX8700.1:BOOL;
	QX8700_2	AT	%QX8700.2:BOOL;
	QX8700_3	AT	%QX8700.3:BOOL;
	QX8700_4	AT	%QX8700.4:BOOL;
	QX8700_5_码垛区域1上托盘按钮指示灯	AT	%QX8700.5:BOOL;
	QX8700_6_码垛区域1下托盘按钮指示灯	AT	%QX8700.6:BOOL;
	QX8700_7	AT	%QX8700.7:BOOL;
	QX8701_0	AT	%QX8701.0:BOOL;
	QX8701_1_码垛区域2上托盘按钮指示灯	AT	%QX8701.1:BOOL;
	QX8701_2_码垛区域2下托盘按钮指示灯	AT	%QX8701.2:BOOL;
	QX8701_3	AT	%QX8701.3:BOOL;
	QX8701_4	AT	%QX8701.4:BOOL;
	QX8701_5_码垛区域3上托盘按钮指示灯	AT	%QX8701.5:BOOL;
	QX8701_6_码垛区域3下托盘按钮指示灯	AT	%QX8701.6:BOOL;
	QX8701_7	AT	%QX8701.7:BOOL;
END_VAR
(* ==== End of DB80_IO ==== *)

(* ---- Main_Clock.st ---- *)
VAR_GLOBAL
	CPU_Clock:Str_Clock;
END_VAR

(* ---- Main_Communication.st ---- *)
VAR_GLOBAL
	From_OPXX AT %IW2000:Str_OP10_TO_OPXX;
	TO_OPXX AT %QW2000:Str_OPXX_TO_OP10;
	To_Slave:Str_ToSlave;

END_VAR
